Yaskawa INFORM job: DEMO_ROOF_UPPER_0625_3PAINT_40.JBI

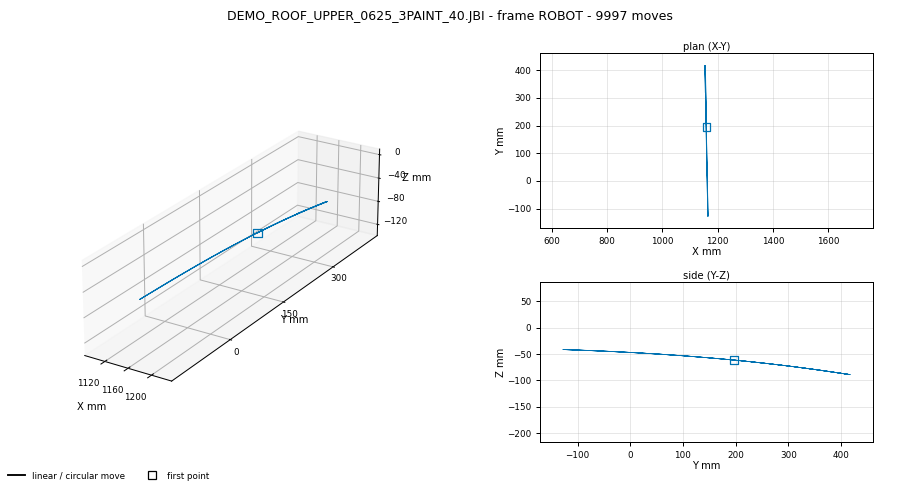
[picture p0: tool path of DEMO_ROOF_UPPER_0625_3PAINT_40.JBI in frame ROBOT, 9997 of 9997 moves have a stored position in this frame; points joined in program order, loops and branches not executed]
/JOB
//NAME DEMO_ROOF_UPPER_0625_3PAINT40
//POS
///NPOS 9997,0,0,0,0,0
///TOOL 0
///USER 0
///POSTYPE ROBOT
///RECTAN
///RCONF 1,0,0,0,0,0,0,0,0,0,0,0,0,0,0,0,0,0,0,0,0,0,0,0
C00000=1159.297,196.712,-61.157,-178.041,7.113,148.757
C00001=1159.293,196.961,-61.181,-178.039,7.115,148.757
C00002=1159.289,197.210,-61.205,-178.035,7.118,148.757
C00003=1159.284,197.459,-61.229,-178.033,7.120,148.756
C00004=1159.280,197.708,-61.253,-178.030,7.122,148.756
C00005=1159.275,197.956,-61.277,-178.027,7.124,148.756
C00006=1159.271,198.205,-61.300,-178.024,7.127,148.756
C00007=1159.265,198.454,-61.325,-178.022,7.129,148.756
C00008=1159.261,198.702,-61.349,-178.019,7.131,148.755
C00009=1159.257,198.952,-61.372,-178.016,7.134,148.755
C00010=1159.252,199.201,-61.396,-178.013,7.135,148.755
C00011=1159.248,199.450,-61.420,-178.011,7.138,148.755
C00012=1159.243,199.698,-61.445,-178.008,7.140,148.754
C00013=1159.238,199.947,-61.469,-178.005,7.143,148.754
C00014=1159.234,200.195,-61.493,-178.003,7.145,148.754
C00015=1159.229,200.444,-61.516,-177.999,7.147,148.754
C00016=1159.225,200.694,-61.541,-177.997,7.149,148.753
C00017=1159.220,200.942,-61.565,-177.994,7.152,148.753
C00018=1159.216,201.191,-61.588,-177.992,7.154,148.753
C00019=1159.211,201.439,-61.613,-177.989,7.156,148.753
C00020=1159.206,201.688,-61.637,-177.986,7.159,148.752
C00021=1159.202,201.937,-61.662,-177.983,7.161,148.752
C00022=1159.198,202.186,-61.685,-177.981,7.164,148.752
C00023=1159.192,202.435,-61.710,-177.978,7.165,148.752
C00024=1159.188,202.683,-61.734,-177.975,7.168,148.751
C00025=1159.184,202.933,-61.758,-177.973,7.170,148.751
C00026=1159.179,203.181,-61.783,-177.969,7.173,148.751
C00027=1159.175,203.430,-61.807,-177.967,7.175,148.751
C00028=1159.170,203.679,-61.830,-177.964,7.177,148.750
C00029=1159.165,203.928,-61.855,-177.962,7.179,148.750
C00030=1159.161,204.177,-61.879,-177.958,7.182,148.750
C00031=1159.157,204.425,-61.903,-177.956,7.184,148.750
C00032=1159.152,204.674,-61.928,-177.953,7.187,148.750
C00033=1159.148,204.923,-61.953,-177.951,7.189,148.749
C00034=1159.143,205.171,-61.977,-177.947,7.191,148.749
C00035=1159.138,205.420,-62.001,-177.945,7.193,148.749
C00036=1159.134,205.668,-62.025,-177.942,7.196,148.749
C00037=1159.129,205.918,-62.050,-177.940,7.198,148.749
C00038=1159.125,206.166,-62.075,-177.937,7.201,148.748
C00039=1159.120,206.415,-62.099,-177.934,7.203,148.748
C00040=1159.116,206.664,-62.124,-177.931,7.205,148.748
C00041=1159.111,206.913,-62.148,-177.929,7.208,148.748
C00042=1159.106,207.161,-62.172,-177.926,7.210,148.747
C00043=1159.101,207.410,-62.197,-177.923,7.212,148.747
C00044=1159.098,207.659,-62.221,-177.920,7.215,148.747
C00045=1159.093,207.907,-62.246,-177.918,7.217,148.747
C00046=1159.088,208.156,-62.270,-177.915,7.220,148.746
C00047=1159.083,208.406,-62.295,-177.913,7.222,148.746
C00048=1159.079,208.654,-62.319,-177.909,7.224,148.746
C00049=1159.074,208.903,-62.344,-177.907,7.226,148.746
C00050=1159.070,209.152,-62.368,-177.904,7.229,148.746
C00051=1159.065,209.400,-62.394,-177.902,7.231,148.745
C00052=1159.060,209.671,-62.420,-177.898,7.234,148.745
C00053=1159.055,209.942,-62.447,-177.895,7.236,148.745
C00054=1159.050,210.212,-62.474,-177.892,7.239,148.745
C00055=1159.046,210.483,-62.501,-177.889,7.242,148.744
C00056=1159.041,210.731,-62.525,-177.887,7.244,148.744
C00057=1159.037,210.980,-62.551,-177.884,7.246,148.744
C00058=1159.033,211.228,-62.575,-177.881,7.249,148.744
C00059=1159.027,211.477,-62.599,-177.878,7.251,148.744
C00060=1159.023,211.726,-62.624,-177.876,7.253,148.743
C00061=1159.019,211.974,-62.649,-177.873,7.256,148.743
C00062=1159.014,212.224,-62.674,-177.870,7.258,148.743
C00063=1159.009,212.472,-62.699,-177.867,7.261,148.743
C00064=1159.006,212.721,-62.724,-177.865,7.263,148.743
C00065=1159.001,212.970,-62.749,-177.862,7.266,148.742
C00066=1158.995,213.218,-62.773,-177.859,7.268,148.742
C00067=1158.992,213.467,-62.798,-177.857,7.270,148.742
C00068=1158.987,213.716,-62.823,-177.854,7.273,148.742
C00069=1158.982,213.965,-62.848,-177.851,7.275,148.742
C00070=1158.978,214.213,-62.873,-177.848,7.278,148.741
C00071=1158.974,214.462,-62.898,-177.846,7.280,148.741
C00072=1158.969,214.711,-62.923,-177.843,7.282,148.741
C00073=1158.965,214.959,-62.948,-177.840,7.284,148.741
C00074=1158.960,215.208,-62.972,-177.838,7.287,148.741
C00075=1158.956,215.457,-62.998,-177.834,7.290,148.740
C00076=1158.951,215.706,-63.023,-177.832,7.292,148.740
C00077=1158.947,215.954,-63.048,-177.829,7.295,148.740
C00078=1158.942,216.203,-63.073,-177.827,7.297,148.740
C00079=1158.938,216.452,-63.098,-177.823,7.299,148.739
C00080=1158.933,216.700,-63.123,-177.821,7.301,148.739
C00081=1158.928,216.949,-63.149,-177.819,7.304,148.739
C00082=1158.924,217.198,-63.173,-177.815,7.307,148.739
C00083=1158.920,217.446,-63.199,-177.813,7.309,148.739
C00084=1158.915,217.695,-63.223,-177.810,7.312,148.738
C00085=1158.910,217.944,-63.249,-177.808,7.314,148.738
C00086=1158.905,218.193,-63.274,-177.805,7.317,148.738
C00087=1158.902,218.441,-63.299,-177.802,7.319,148.738
C00088=1158.897,218.689,-63.324,-177.799,7.321,148.738
C00089=1158.892,218.939,-63.349,-177.796,7.324,148.738
C00090=1158.888,219.187,-63.375,-177.794,7.326,148.737
C00091=1158.883,219.436,-63.401,-177.791,7.329,148.737
C00092=1158.879,219.685,-63.426,-177.788,7.332,148.737
C00093=1158.874,219.933,-63.451,-177.786,7.334,148.737
C00094=1158.871,220.182,-63.476,-177.782,7.336,148.737
C00095=1158.865,220.430,-63.501,-177.780,7.338,148.736
C00096=1158.861,220.679,-63.527,-177.777,7.341,148.736
C00097=1158.857,220.928,-63.552,-177.774,7.344,148.736
C00098=1158.852,221.177,-63.577,-177.772,7.346,148.736
C00099=1158.848,221.425,-63.603,-177.769,7.349,148.736
C00100=1158.843,221.674,-63.628,-177.767,7.351,148.736
C00101=1158.839,221.922,-63.654,-177.764,7.354,148.735
C00102=1158.834,222.171,-63.680,-177.761,7.356,148.735
C00103=1158.829,222.420,-63.704,-177.758,7.358,148.735
C00104=1158.825,222.669,-63.730,-177.756,7.361,148.735
C00105=1158.821,222.918,-63.756,-177.752,7.364,148.735
C00106=1158.816,223.166,-63.781,-177.750,7.366,148.735
C00107=1158.812,223.414,-63.807,-177.747,7.369,148.734
C00108=1158.807,223.663,-63.832,-177.744,7.372,148.734
C00109=1158.802,223.912,-63.857,-177.742,7.374,148.734
C00110=1158.798,224.161,-63.883,-177.739,7.376,148.734
C00111=1158.793,224.409,-63.908,-177.736,7.378,148.734
C00112=1158.789,224.658,-63.934,-177.734,7.381,148.734
C00113=1158.785,224.906,-63.960,-177.730,7.384,148.733
C00114=1158.781,225.155,-63.986,-177.728,7.386,148.733
C00115=1158.776,225.403,-64.011,-177.725,7.389,148.733
C00116=1158.772,225.652,-64.037,-177.722,7.392,148.733
C00117=1158.767,225.901,-64.063,-177.720,7.394,148.733
C00118=1158.762,226.149,-64.088,-177.717,7.397,148.732
C00119=1158.758,226.398,-64.114,-177.714,7.399,148.732
C00120=1158.753,226.647,-64.140,-177.712,7.401,148.732
C00121=1158.748,226.895,-64.165,-177.709,7.404,148.732
C00122=1158.744,227.144,-64.191,-177.706,7.407,148.732
C00123=1158.740,227.393,-64.217,-177.704,7.409,148.732
C00124=1158.736,227.642,-64.243,-177.701,7.412,148.731
C00125=1158.731,227.890,-64.268,-177.698,7.415,148.731
C00126=1158.726,228.139,-64.294,-177.695,7.417,148.731
C00127=1158.722,228.388,-64.320,-177.693,7.420,148.731
C00128=1158.718,228.636,-64.346,-177.690,7.423,148.731
C00129=1158.713,228.884,-64.371,-177.687,7.424,148.731
C00130=1158.709,229.133,-64.398,-177.684,7.427,148.731
C00131=1158.705,229.381,-64.424,-177.682,7.430,148.730
C00132=1158.700,229.631,-64.450,-177.679,7.432,148.730
C00133=1158.695,229.879,-64.476,-177.676,7.435,148.730
C00134=1158.691,230.127,-64.501,-177.673,7.438,148.730
C00135=1158.686,230.376,-64.527,-177.671,7.440,148.730
C00136=1158.682,230.625,-64.554,-177.668,7.443,148.730
C00137=1158.677,230.874,-64.580,-177.665,7.446,148.729
C00138=1158.673,231.122,-64.605,-177.663,7.448,148.729
C00139=1158.668,231.370,-64.631,-177.660,7.450,148.729
C00140=1158.664,231.619,-64.658,-177.657,7.453,148.729
C00141=1158.660,231.868,-64.684,-177.654,7.456,148.729
C00142=1158.655,232.117,-64.709,-177.651,7.458,148.729
C00143=1158.651,232.365,-64.736,-177.649,7.461,148.728
C00144=1158.646,232.613,-64.762,-177.646,7.464,148.728
C00145=1158.642,232.862,-64.787,-177.644,7.466,148.728
C00146=1158.637,233.110,-64.815,-177.640,7.468,148.728
C00147=1158.633,233.359,-64.840,-177.638,7.471,148.728
C00148=1158.628,233.608,-64.866,-177.635,7.474,148.728
C00149=1158.624,233.857,-64.893,-177.633,7.476,148.728
C00150=1158.620,234.105,-64.919,-177.630,7.479,148.727
C00151=1158.615,234.354,-64.945,-177.627,7.482,148.727
C00152=1158.610,234.602,-64.971,-177.625,7.484,148.727
C00153=1158.606,234.851,-64.997,-177.622,7.487,148.727
C00154=1158.601,235.099,-65.024,-177.619,7.490,148.727
C00155=1158.597,235.348,-65.050,-177.616,7.493,148.727
C00156=1158.593,235.619,-65.079,-177.613,7.496,148.727
C00157=1158.587,235.892,-65.107,-177.610,7.498,148.726
C00158=1158.583,236.163,-65.136,-177.607,7.501,148.726
C00159=1158.578,236.434,-65.165,-177.604,7.504,148.726
C00160=1158.573,236.683,-65.191,-177.601,7.507,148.726
C00161=1158.569,236.932,-65.218,-177.599,7.509,148.726
C00162=1158.565,237.181,-65.244,-177.596,7.512,148.726
C00163=1158.560,237.429,-65.271,-177.593,7.515,148.726
C00164=1158.556,237.678,-65.297,-177.590,7.518,148.726
C00165=1158.551,237.926,-65.324,-177.588,7.519,148.725
C00166=1158.547,238.175,-65.350,-177.585,7.522,148.725
C00167=1158.542,238.424,-65.377,-177.582,7.525,148.725
C00168=1158.538,238.672,-65.403,-177.579,7.528,148.725
C00169=1158.534,238.920,-65.430,-177.577,7.530,148.725
C00170=1158.529,239.169,-65.456,-177.574,7.533,148.725
C00171=1158.525,239.418,-65.483,-177.571,7.536,148.725
C00172=1158.520,239.666,-65.510,-177.568,7.539,148.725
C00173=1158.516,239.915,-65.536,-177.566,7.541,148.724
C00174=1158.511,240.163,-65.563,-177.563,7.544,148.724
C00175=1158.507,240.412,-65.589,-177.560,7.546,148.724
C00176=1158.502,240.661,-65.616,-177.557,7.549,148.724
C00177=1158.498,240.909,-65.642,-177.555,7.552,148.724
C00178=1158.494,241.157,-65.669,-177.553,7.554,148.724
C00179=1158.489,241.406,-65.696,-177.550,7.557,148.724
C00180=1158.485,241.655,-65.722,-177.547,7.560,148.723
C00181=1158.480,241.903,-65.749,-177.544,7.562,148.723
C00182=1158.476,242.152,-65.776,-177.542,7.565,148.723
C00183=1158.472,242.400,-65.803,-177.539,7.568,148.723
C00184=1158.467,242.648,-65.830,-177.536,7.571,148.723
C00185=1158.462,242.897,-65.857,-177.533,7.574,148.723
C00186=1158.458,243.146,-65.882,-177.531,7.576,148.723
C00187=1158.453,243.394,-65.910,-177.528,7.579,148.723
C00188=1158.449,243.643,-65.937,-177.525,7.582,148.723
C00189=1158.445,243.891,-65.963,-177.522,7.585,148.722
C00190=1158.440,244.139,-65.990,-177.519,7.587,148.722
C00191=1158.436,244.389,-66.018,-177.517,7.590,148.722
C00192=1158.432,244.637,-66.044,-177.514,7.592,148.722
C00193=1158.428,244.885,-66.071,-177.511,7.595,148.722
C00194=1158.423,245.134,-66.098,-177.508,7.598,148.722
C00195=1158.418,245.382,-66.125,-177.506,7.600,148.722
C00196=1158.414,245.630,-66.152,-177.504,7.603,148.722
C00197=1158.410,245.879,-66.179,-177.501,7.606,148.722
C00198=1158.405,246.127,-66.206,-177.498,7.609,148.722
C00199=1158.401,246.377,-66.233,-177.495,7.612,148.721
C00200=1158.396,246.625,-66.260,-177.493,7.614,148.721
C00201=1158.392,246.873,-66.287,-177.490,7.617,148.721
C00202=1158.388,247.122,-66.314,-177.487,7.620,148.721
C00203=1158.383,247.370,-66.341,-177.484,7.623,148.721
C00204=1158.378,247.619,-66.368,-177.481,7.626,148.721
C00205=1158.374,247.867,-66.395,-177.479,7.628,148.721
C00206=1158.370,248.116,-66.423,-177.477,7.631,148.721
C00207=1158.366,248.364,-66.450,-177.474,7.634,148.721
C00208=1158.361,248.613,-66.477,-177.471,7.636,148.720
C00209=1158.357,248.861,-66.504,-177.468,7.639,148.720
C00210=1158.352,249.110,-66.531,-177.465,7.642,148.720
C00211=1158.347,249.358,-66.558,-177.463,7.644,148.720
C00212=1158.344,249.607,-66.586,-177.460,7.647,148.720
C00213=1158.339,249.855,-66.613,-177.457,7.650,148.720
C00214=1158.334,250.104,-66.640,-177.454,7.653,148.720
C00215=1158.330,250.352,-66.667,-177.452,7.656,148.720
C00216=1158.327,250.600,-66.695,-177.449,7.659,148.720
C00217=1158.322,250.849,-66.722,-177.447,7.661,148.720
C00218=1158.317,251.097,-66.749,-177.444,7.664,148.720
C00219=1158.313,251.346,-66.776,-177.441,7.667,148.719
C00220=1158.308,251.594,-66.804,-177.438,7.669,148.719
C00221=1158.304,251.843,-66.831,-177.435,7.672,148.719
C00222=1158.300,252.091,-66.858,-177.432,7.675,148.719
C00223=1158.295,252.339,-66.886,-177.430,7.677,148.719
C00224=1158.291,252.588,-66.913,-177.427,7.680,148.719
C00225=1158.287,252.837,-66.940,-177.425,7.683,148.719
C00226=1158.282,253.085,-66.968,-177.422,7.686,148.719
C00227=1158.278,253.333,-66.995,-177.419,7.689,148.719
C00228=1158.274,253.582,-67.023,-177.416,7.692,148.719
C00229=1158.269,253.830,-67.050,-177.414,7.695,148.719
C00230=1158.265,254.078,-67.078,-177.411,7.697,148.719
C00231=1158.261,254.327,-67.106,-177.409,7.700,148.719
C00232=1158.256,254.576,-67.134,-177.406,7.703,148.718
C00233=1158.251,254.824,-67.161,-177.403,7.706,148.718
C00234=1158.246,255.073,-67.188,-177.400,7.709,148.718
C00235=1158.243,255.321,-67.216,-177.398,7.712,148.718
C00236=1158.238,255.569,-67.244,-177.395,7.715,148.718
C00237=1158.234,255.818,-67.271,-177.393,7.717,148.718
C00238=1158.230,256.066,-67.299,-177.390,7.720,148.718
C00239=1158.225,256.315,-67.326,-177.387,7.723,148.718
C00240=1158.221,256.563,-67.354,-177.384,7.726,148.718
C00241=1158.216,256.812,-67.382,-177.381,7.729,148.718
C00242=1158.212,257.060,-67.410,-177.378,7.731,148.718
C00243=1158.208,257.309,-67.438,-177.376,7.734,148.718
C00244=1158.203,257.557,-67.465,-177.373,7.737,148.717
C00245=1158.199,257.805,-67.493,-177.371,7.739,148.717
C00246=1158.195,258.054,-67.520,-177.368,7.742,148.717
C00247=1158.190,258.302,-67.549,-177.365,7.745,148.717
C00248=1158.185,258.550,-67.576,-177.362,7.748,148.717
C00249=1158.182,258.799,-67.605,-177.360,7.751,148.717
C00250=1158.177,259.047,-67.632,-177.357,7.754,148.717
C00251=1158.173,259.296,-67.660,-177.354,7.757,148.717
C00252=1158.168,259.544,-67.688,-177.351,7.760,148.717
C00253=1158.164,259.792,-67.715,-177.349,7.763,148.717
C00254=1158.160,260.041,-67.743,-177.347,7.766,148.717
C00255=1158.155,260.289,-67.771,-177.344,7.768,148.717
C00256=1158.151,260.538,-67.800,-177.341,7.771,148.717
C00257=1158.147,260.786,-67.828,-177.338,7.774,148.717
C00258=1158.143,261.035,-67.855,-177.336,7.777,148.717
C00259=1158.138,261.283,-67.883,-177.333,7.780,148.717
C00260=1158.133,261.556,-67.914,-177.330,7.783,148.717
C00261=1158.128,261.830,-67.945,-177.327,7.786,148.717
C00262=1158.124,262.102,-67.976,-177.324,7.790,148.717
C00263=1158.119,262.376,-68.007,-177.321,7.793,148.716
C00264=1158.114,262.624,-68.035,-177.318,7.796,148.716
C00265=1158.110,262.873,-68.063,-177.316,7.799,148.716
C00266=1158.106,263.121,-68.090,-177.313,7.802,148.716
C00267=1158.101,263.370,-68.119,-177.310,7.805,148.716
C00268=1158.097,263.618,-68.147,-177.307,7.808,148.716
C00269=1158.093,263.866,-68.175,-177.305,7.811,148.716
C00270=1158.088,264.115,-68.204,-177.302,7.813,148.716
C00271=1158.084,264.363,-68.232,-177.300,7.816,148.716
C00272=1158.079,264.611,-68.260,-177.297,7.819,148.716
C00273=1158.075,264.860,-68.288,-177.294,7.822,148.716
C00274=1158.070,265.108,-68.317,-177.291,7.824,148.716
C00275=1158.067,265.357,-68.345,-177.289,7.827,148.716
C00276=1158.061,265.605,-68.373,-177.286,7.830,148.716
C00277=1158.058,265.853,-68.402,-177.283,7.833,148.716
C00278=1158.054,266.101,-68.430,-177.280,7.836,148.716
C00279=1158.049,266.350,-68.458,-177.278,7.840,148.716
C00280=1158.045,266.598,-68.487,-177.275,7.842,148.716
C00281=1158.040,266.846,-68.515,-177.272,7.845,148.716
C00282=1158.037,267.095,-68.543,-177.270,7.848,148.716
C00283=1158.032,267.343,-68.571,-177.267,7.851,148.716
C00284=1158.027,267.592,-68.600,-177.265,7.853,148.715
C00285=1158.024,267.840,-68.629,-177.262,7.856,148.715
C00286=1158.018,268.088,-68.657,-177.259,7.859,148.715
C00287=1158.015,268.337,-68.686,-177.256,7.862,148.715
C00288=1158.010,268.585,-68.714,-177.254,7.866,148.715
C00289=1158.006,268.833,-68.742,-177.251,7.869,148.715
C00290=1158.002,269.082,-68.772,-177.249,7.871,148.715
C00291=1157.997,269.330,-68.799,-177.246,7.874,148.715
C00292=1157.993,269.579,-68.828,-177.243,7.877,148.715
C00293=1157.988,269.826,-68.857,-177.240,7.880,148.715
C00294=1157.984,270.075,-68.885,-177.238,7.883,148.715
C00295=1157.980,270.324,-68.914,-177.235,7.886,148.715
C00296=1157.976,270.571,-68.942,-177.232,7.890,148.715
C00297=1157.971,270.820,-68.971,-177.230,7.892,148.715
C00298=1157.967,271.069,-69.000,-177.227,7.895,148.715
C00299=1157.963,271.316,-69.028,-177.224,7.898,148.715
C00300=1157.958,271.565,-69.057,-177.221,7.901,148.715
C00301=1157.954,271.814,-69.086,-177.219,7.904,148.715
C00302=1157.950,272.061,-69.114,-177.216,7.907,148.715
C00303=1157.945,272.310,-69.143,-177.214,7.910,148.715
C00304=1157.941,272.558,-69.173,-177.211,7.913,148.715
C00305=1157.937,272.806,-69.200,-177.208,7.916,148.715
C00306=1157.932,273.055,-69.229,-177.205,7.919,148.715
C00307=1157.928,273.303,-69.259,-177.203,7.921,148.715
C00308=1157.924,273.552,-69.287,-177.200,7.924,148.715
C00309=1157.920,273.799,-69.316,-177.198,7.928,148.715
C00310=1157.915,274.048,-69.345,-177.195,7.931,148.715
C00311=1157.911,274.296,-69.374,-177.192,7.934,148.715
C00312=1157.906,274.544,-69.403,-177.190,7.937,148.715
C00313=1157.902,274.792,-69.431,-177.187,7.940,148.715
C00314=1157.898,275.041,-69.461,-177.185,7.943,148.715
C00315=1157.894,275.290,-69.489,-177.182,7.946,148.715
C00316=1157.889,275.537,-69.519,-177.179,7.949,148.715
C00317=1157.884,275.786,-69.547,-177.176,7.952,148.715
C00318=1157.881,276.034,-69.576,-177.174,7.955,148.715
C00319=1157.877,276.282,-69.606,-177.171,7.958,148.715
C00320=1157.872,276.531,-69.634,-177.169,7.961,148.715
C00321=1157.868,276.779,-69.663,-177.166,7.964,148.715
C00322=1157.863,277.027,-69.693,-177.163,7.967,148.715
C00323=1157.859,277.276,-69.722,-177.160,7.970,148.715
C00324=1157.855,277.524,-69.750,-177.158,7.973,148.715
C00325=1157.851,277.771,-69.780,-177.155,7.976,148.715
C00326=1157.846,278.020,-69.809,-177.152,7.979,148.715
C00327=1157.842,278.269,-69.838,-177.150,7.982,148.715
C00328=1157.838,278.517,-69.867,-177.147,7.985,148.715
C00329=1157.834,278.765,-69.897,-177.145,7.988,148.715
C00330=1157.829,279.013,-69.926,-177.142,7.991,148.715
C00331=1157.824,279.262,-69.954,-177.139,7.994,148.715
C00332=1157.820,279.510,-69.984,-177.137,7.997,148.715
C00333=1157.817,279.758,-70.013,-177.134,8.000,148.715
C00334=1157.813,280.006,-70.042,-177.131,8.003,148.715
C00335=1157.808,280.254,-70.072,-177.128,8.006,148.715
C00336=1157.804,280.503,-70.101,-177.126,8.009,148.715
C00337=1157.800,280.751,-70.131,-177.123,8.012,148.715
C00338=1157.795,280.999,-70.159,-177.121,8.015,148.715
C00339=1157.791,281.247,-70.188,-177.118,8.018,148.715
C00340=1157.787,281.496,-70.218,-177.116,8.022,148.715
C00341=1157.782,281.744,-70.247,-177.113,8.024,148.715
C00342=1157.778,281.992,-70.277,-177.110,8.027,148.715
C00343=1157.774,282.240,-70.306,-177.107,8.031,148.715
C00344=1157.769,282.489,-70.336,-177.104,8.034,148.715
C00345=1157.765,282.737,-70.366,-177.102,8.037,148.715
C00346=1157.761,282.986,-70.395,-177.099,8.040,148.715
C00347=1157.756,283.233,-70.424,-177.097,8.044,148.715
C00348=1157.752,283.481,-70.454,-177.094,8.047,148.715
C00349=1157.748,283.730,-70.483,-177.091,8.050,148.715
C00350=1157.743,283.978,-70.513,-177.088,8.053,148.715
C00351=1157.739,284.226,-70.542,-177.086,8.056,148.715
C00352=1157.735,284.474,-70.572,-177.083,8.059,148.715
C00353=1157.731,284.723,-70.601,-177.080,8.062,148.715
C00354=1157.727,284.971,-70.630,-177.078,8.065,148.715
C00355=1157.722,285.219,-70.661,-177.075,8.068,148.715
C00356=1157.718,285.467,-70.691,-177.073,8.071,148.715
C00357=1157.714,285.715,-70.720,-177.070,8.074,148.715
C00358=1157.709,285.964,-70.750,-177.068,8.077,148.715
C00359=1157.705,286.212,-70.779,-177.065,8.080,148.715
C00360=1157.701,286.460,-70.808,-177.062,8.083,148.715
C00361=1157.697,286.708,-70.839,-177.060,8.086,148.715
C00362=1157.692,286.956,-70.869,-177.057,8.089,148.715
C00363=1157.688,287.205,-70.898,-177.055,8.093,148.716
C00364=1157.684,287.480,-70.931,-177.051,8.096,148.716
C00365=1157.679,287.755,-70.964,-177.049,8.099,148.716
C00366=1157.674,288.030,-70.997,-177.045,8.103,148.716
C00367=1157.669,288.305,-71.030,-177.043,8.106,148.716
C00368=1157.665,288.553,-71.060,-177.040,8.109,148.716
C00369=1157.660,288.801,-71.090,-177.037,8.112,148.716
C00370=1157.656,289.050,-71.120,-177.034,8.116,148.716
C00371=1157.652,289.297,-71.150,-177.032,8.119,148.716
C00372=1157.648,289.545,-71.179,-177.029,8.123,148.716
C00373=1157.644,289.795,-71.210,-177.027,8.126,148.716
C00374=1157.640,290.042,-71.240,-177.024,8.128,148.716
C00375=1157.636,290.291,-71.269,-177.022,8.132,148.716
C00376=1157.631,290.539,-71.300,-177.019,8.135,148.716
C00377=1157.627,290.787,-71.330,-177.016,8.138,148.716
C00378=1157.623,291.035,-71.359,-177.014,8.141,148.716
C00379=1157.618,291.283,-71.390,-177.011,8.144,148.716
C00380=1157.614,291.531,-71.419,-177.009,8.147,148.716
C00381=1157.610,291.779,-71.449,-177.006,8.150,148.716
C00382=1157.605,292.028,-71.479,-177.003,8.153,148.716
C00383=1157.601,292.275,-71.510,-177.000,8.157,148.716
C00384=1157.598,292.524,-71.539,-176.998,8.160,148.716
C00385=1157.593,292.772,-71.570,-176.995,8.163,148.717
C00386=1157.589,293.020,-71.600,-176.992,8.166,148.717
C00387=1157.584,293.268,-71.630,-176.990,8.169,148.717
C00388=1157.580,293.516,-71.661,-176.987,8.173,148.717
C00389=1157.575,293.765,-71.691,-176.985,8.176,148.717
C00390=1157.571,294.012,-71.721,-176.982,8.179,148.717
C00391=1157.568,294.261,-71.751,-176.980,8.182,148.717
C00392=1157.563,294.509,-71.781,-176.977,8.185,148.717
C00393=1157.559,294.757,-71.812,-176.975,8.188,148.717
C00394=1157.554,295.005,-71.842,-176.971,8.192,148.717
C00395=1157.551,295.253,-71.872,-176.969,8.195,148.717
C00396=1157.546,295.501,-71.903,-176.966,8.198,148.717
C00397=1157.542,295.750,-71.932,-176.964,8.201,148.717
C00398=1157.538,295.998,-71.963,-176.961,8.204,148.717
C00399=1157.534,296.246,-71.993,-176.959,8.208,148.717
C00400=1157.529,296.494,-72.024,-176.956,8.211,148.717
C00401=1157.525,296.742,-72.053,-176.953,8.213,148.717
C00402=1157.521,296.990,-72.085,-176.951,8.217,148.718
C00403=1157.517,297.238,-72.115,-176.948,8.220,148.718
C00404=1157.513,297.486,-72.146,-176.945,8.224,148.718
C00405=1157.508,297.734,-72.176,-176.943,8.227,148.718
C00406=1157.504,297.983,-72.206,-176.940,8.230,148.718
C00407=1157.500,298.231,-72.237,-176.937,8.233,148.718
C00408=1157.496,298.479,-72.267,-176.935,8.236,148.718
C00409=1157.491,298.727,-72.298,-176.932,8.239,148.718
C00410=1157.487,298.975,-72.329,-176.930,8.243,148.718
C00411=1157.483,299.223,-72.359,-176.927,8.246,148.718
C00412=1157.479,299.471,-72.390,-176.924,8.250,148.718
C00413=1157.474,299.719,-72.421,-176.922,8.253,148.718
C00414=1157.471,299.968,-72.450,-176.919,8.256,148.719
C00415=1157.466,300.216,-72.481,-176.917,8.259,148.718
C00416=1157.461,300.464,-72.512,-176.914,8.262,148.719
C00417=1157.458,300.711,-72.542,-176.912,8.265,148.719
C00418=1157.454,300.960,-72.573,-176.909,8.268,148.719
C00419=1157.449,301.208,-72.604,-176.906,8.271,148.719
C00420=1157.445,301.456,-72.634,-176.904,8.275,148.719
C00421=1157.441,301.704,-72.665,-176.901,8.278,148.719
C00422=1157.436,301.952,-72.696,-176.899,8.282,148.719
C00423=1157.432,302.200,-72.728,-176.896,8.285,148.719
C00424=1157.429,302.448,-72.758,-176.893,8.288,148.719
C00425=1157.424,302.696,-72.789,-176.891,8.291,148.719
C00426=1157.420,302.944,-72.820,-176.888,8.294,148.719
C00427=1157.416,303.192,-72.851,-176.885,8.298,148.719
C00428=1157.412,303.440,-72.881,-176.883,8.301,148.720
C00429=1157.407,303.688,-72.912,-176.880,8.304,148.720
C00430=1157.403,303.937,-72.943,-176.878,8.307,148.720
C00431=1157.398,304.185,-72.974,-176.875,8.311,148.720
C00432=1157.394,304.432,-73.005,-176.873,8.314,148.720
C00433=1157.390,304.681,-73.036,-176.870,8.318,148.720
C00434=1157.386,304.928,-73.066,-176.867,8.321,148.720
C00435=1157.382,305.177,-73.098,-176.865,8.324,148.720
C00436=1157.378,305.424,-73.129,-176.862,8.327,148.720
C00437=1157.373,305.672,-73.160,-176.860,8.330,148.720
C00438=1157.369,305.921,-73.191,-176.857,8.333,148.721
C00439=1157.365,306.169,-73.222,-176.854,8.337,148.721
C00440=1157.361,306.417,-73.254,-176.852,8.341,148.721
C00441=1157.356,306.665,-73.284,-176.849,8.344,148.721
C00442=1157.353,306.913,-73.314,-176.847,8.347,148.721
C00443=1157.349,307.161,-73.346,-176.844,8.350,148.721
C00444=1157.344,307.409,-73.377,-176.842,8.353,148.721
C00445=1157.340,307.657,-73.408,-176.839,8.357,148.721
C00446=1157.336,307.905,-73.440,-176.836,8.360,148.721
C00447=1157.332,308.153,-73.471,-176.834,8.363,148.722
C00448=1157.327,308.401,-73.502,-176.831,8.366,148.722
C00449=1157.323,308.648,-73.533,-176.829,8.370,148.722
C00450=1157.319,308.897,-73.564,-176.826,8.373,148.722
C00451=1157.315,309.144,-73.596,-176.823,8.377,148.722
C00452=1157.311,309.393,-73.627,-176.821,8.380,148.722
C00453=1157.306,309.640,-73.658,-176.818,8.383,148.722
C00454=1157.302,309.889,-73.689,-176.816,8.386,148.722
C00455=1157.298,310.136,-73.721,-176.813,8.389,148.722
C00456=1157.294,310.385,-73.752,-176.810,8.393,148.723
C00457=1157.290,310.632,-73.783,-176.808,8.397,148.723
C00458=1157.286,310.881,-73.815,-176.805,8.400,148.723
C00459=1157.281,311.128,-73.846,-176.803,8.403,148.723
C00460=1157.277,311.377,-73.877,-176.800,8.406,148.723
C00461=1157.273,311.624,-73.909,-176.797,8.410,148.723
C00462=1157.269,311.873,-73.941,-176.795,8.413,148.723
C00463=1157.265,312.120,-73.971,-176.792,8.416,148.723
C00464=1157.260,312.369,-74.004,-176.789,8.419,148.723
C00465=1157.256,312.617,-74.035,-176.787,8.423,148.724
C00466=1157.252,312.865,-74.066,-176.784,8.427,148.724
C00467=1157.248,313.113,-74.098,-176.782,8.430,148.724
C00468=1157.243,313.390,-74.133,-176.779,8.433,148.724
C00469=1157.239,313.668,-74.168,-176.776,8.437,148.724
C00470=1157.234,313.945,-74.204,-176.773,8.441,148.724
C00471=1157.229,314.222,-74.239,-176.770,8.445,148.724
C00472=1157.225,314.470,-74.271,-176.768,8.448,148.725
C00473=1157.221,314.718,-74.303,-176.765,8.451,148.725
C00474=1157.217,314.966,-74.334,-176.763,8.454,148.725
C00475=1157.212,315.214,-74.366,-176.760,8.458,148.725
C00476=1157.209,315.462,-74.398,-176.757,8.462,148.725
C00477=1157.204,315.709,-74.429,-176.755,8.465,148.725
C00478=1157.201,315.957,-74.461,-176.753,8.468,148.725
C00479=1157.196,316.206,-74.493,-176.750,8.471,148.726
C00480=1157.192,316.454,-74.524,-176.747,8.475,148.726
C00481=1157.188,316.702,-74.556,-176.745,8.478,148.726
C00482=1157.184,316.950,-74.588,-176.742,8.482,148.726
C00483=1157.180,317.197,-74.619,-176.739,8.485,148.726
C00484=1157.175,317.445,-74.652,-176.737,8.488,148.726
C00485=1157.172,317.693,-74.684,-176.734,8.492,148.726
C00486=1157.167,317.941,-74.715,-176.732,8.495,148.727
C00487=1157.163,318.189,-74.747,-176.729,8.498,148.727
C00488=1157.159,318.437,-74.779,-176.727,8.502,148.727
C00489=1157.155,318.684,-74.811,-176.724,8.506,148.727
C00490=1157.151,318.933,-74.843,-176.722,8.509,148.727
C00491=1157.147,319.181,-74.875,-176.719,8.512,148.727
C00492=1157.143,319.428,-74.907,-176.717,8.515,148.727
C00493=1157.138,319.677,-74.939,-176.714,8.519,148.728
C00494=1157.134,319.925,-74.971,-176.711,8.523,148.728
C00495=1157.131,320.173,-75.003,-176.709,8.526,148.728
C00496=1157.126,320.420,-75.035,-176.706,8.529,148.728
C00497=1157.122,320.668,-75.067,-176.704,8.533,148.728
C00498=1157.118,320.916,-75.098,-176.701,8.536,148.728
C00499=1157.114,321.165,-75.131,-176.698,8.539,148.728
C00500=1157.109,321.412,-75.162,-176.696,8.542,148.729
C00501=1157.105,321.660,-75.196,-176.693,8.547,148.729
C00502=1157.102,321.908,-75.227,-176.691,8.550,148.729
C00503=1157.098,322.156,-75.259,-176.688,8.553,148.729
C00504=1157.093,322.403,-75.291,-176.686,8.556,148.729
C00505=1157.089,322.652,-75.323,-176.683,8.560,148.729
C00506=1157.085,322.899,-75.356,-176.681,8.563,148.730
C00507=1157.081,323.147,-75.388,-176.678,8.567,148.730
C00508=1157.076,323.395,-75.420,-176.676,8.570,148.730
C00509=1157.073,323.643,-75.452,-176.673,8.574,148.730
C00510=1157.068,323.891,-75.485,-176.670,8.577,148.730
C00511=1157.065,324.139,-75.517,-176.668,8.580,148.730
C00512=1157.060,324.387,-75.549,-176.665,8.584,148.731
C00513=1157.056,324.634,-75.582,-176.663,8.588,148.731
C00514=1157.052,324.882,-75.614,-176.660,8.591,148.731
C00515=1157.048,325.130,-75.646,-176.658,8.594,148.731
C00516=1157.044,325.378,-75.679,-176.655,8.598,148.731
C00517=1157.040,325.626,-75.711,-176.653,8.601,148.732
C00518=1157.036,325.874,-75.743,-176.650,8.605,148.732
C00519=1157.031,326.121,-75.776,-176.647,8.609,148.732
C00520=1157.027,326.369,-75.808,-176.645,8.612,148.732
C00521=1157.023,326.617,-75.841,-176.642,8.615,148.732
C00522=1157.020,326.865,-75.873,-176.640,8.618,148.732
C00523=1157.015,327.114,-75.905,-176.637,8.622,148.733
C00524=1157.011,327.361,-75.939,-176.635,8.626,148.733
C00525=1157.007,327.609,-75.970,-176.633,8.629,148.733
C00526=1157.003,327.856,-76.003,-176.630,8.633,148.733
C00527=1156.998,328.105,-76.036,-176.627,8.636,148.733
C00528=1156.995,328.352,-76.068,-176.625,8.639,148.733
C00529=1156.991,328.600,-76.101,-176.622,8.643,148.734
C00530=1156.986,328.848,-76.134,-176.619,8.647,148.734
C00531=1156.983,329.096,-76.166,-176.617,8.650,148.734
C00532=1156.978,329.344,-76.199,-176.615,8.653,148.734
C00533=1156.974,329.592,-76.232,-176.612,8.657,148.734
C00534=1156.970,329.840,-76.264,-176.610,8.661,148.735
C00535=1156.966,330.087,-76.297,-176.607,8.664,148.735
C00536=1156.962,330.335,-76.330,-176.604,8.668,148.735
C00537=1156.957,330.583,-76.362,-176.602,8.671,148.735
C00538=1156.954,330.830,-76.395,-176.599,8.674,148.735
C00539=1156.950,331.078,-76.428,-176.597,8.678,148.736
C00540=1156.945,331.326,-76.460,-176.594,8.682,148.736
C00541=1156.941,331.574,-76.494,-176.592,8.685,148.736
C00542=1156.938,331.821,-76.526,-176.589,8.689,148.736
C00543=1156.933,332.069,-76.559,-176.587,8.692,148.736
C00544=1156.929,332.318,-76.592,-176.584,8.696,148.737
C00545=1156.925,332.565,-76.625,-176.581,8.700,148.737
C00546=1156.921,332.813,-76.658,-176.579,8.703,148.737
C00547=1156.917,333.061,-76.691,-176.577,8.706,148.737
C00548=1156.913,333.308,-76.724,-176.574,8.710,148.737
C00549=1156.909,333.556,-76.756,-176.571,8.713,148.737
C00550=1156.905,333.804,-76.789,-176.569,8.717,148.738
C00551=1156.900,334.052,-76.823,-176.566,8.721,148.738
C00552=1156.896,334.300,-76.856,-176.564,8.724,148.738
C00553=1156.892,334.547,-76.889,-176.561,8.727,148.738
C00554=1156.888,334.795,-76.922,-176.559,8.731,148.739
C00555=1156.885,335.043,-76.955,-176.556,8.735,148.739
C00556=1156.880,335.290,-76.988,-176.554,8.738,148.739
C00557=1156.876,335.538,-77.021,-176.551,8.742,148.739
C00558=1156.872,335.786,-77.054,-176.549,8.745,148.739
C00559=1156.868,336.034,-77.086,-176.546,8.749,148.740
C00560=1156.864,336.282,-77.120,-176.544,8.753,148.740
C00561=1156.860,336.530,-77.153,-176.541,8.756,148.740
C00562=1156.856,336.778,-77.186,-176.539,8.759,148.740
C00563=1156.852,337.025,-77.220,-176.536,8.763,148.741
C00564=1156.848,337.273,-77.253,-176.534,8.767,148.741
C00565=1156.844,337.521,-77.286,-176.531,8.770,148.741
C00566=1156.840,337.768,-77.320,-176.528,8.774,148.741
C00567=1156.836,338.016,-77.353,-176.526,8.777,148.741
C00568=1156.831,338.264,-77.386,-176.523,8.781,148.742
C00569=1156.827,338.511,-77.419,-176.521,8.785,148.742
C00570=1156.823,338.759,-77.452,-176.519,8.788,148.742
C00571=1156.820,339.008,-77.486,-176.516,8.792,148.742
C00572=1156.815,339.287,-77.523,-176.513,8.796,148.743
C00573=1156.810,339.567,-77.561,-176.510,8.800,148.743
C00574=1156.805,339.847,-77.599,-176.508,8.804,148.743
C00575=1156.801,340.127,-77.637,-176.505,8.808,148.743
C00576=1156.797,340.375,-77.670,-176.502,8.812,148.744
C00577=1156.793,340.622,-77.703,-176.500,8.815,148.744
C00578=1156.789,340.870,-77.737,-176.497,8.819,148.744
C00579=1156.785,341.117,-77.770,-176.495,8.823,148.744
C00580=1156.780,341.365,-77.804,-176.493,8.826,148.745
C00581=1156.776,341.614,-77.837,-176.490,8.830,148.745
C00582=1156.773,341.861,-77.871,-176.487,8.833,148.745
C00583=1156.768,342.109,-77.904,-176.484,8.837,148.745
C00584=1156.764,342.356,-77.938,-176.482,8.841,148.745
C00585=1156.760,342.603,-77.972,-176.480,8.844,148.746
C00586=1156.756,342.851,-78.005,-176.477,8.848,148.746
C00587=1156.752,343.099,-78.040,-176.475,8.851,148.746
C00588=1156.748,343.347,-78.073,-176.472,8.856,148.746
C00589=1156.744,343.595,-78.106,-176.469,8.859,148.747
C00590=1156.740,343.842,-78.140,-176.467,8.862,148.747
C00591=1156.736,344.091,-78.174,-176.465,8.866,148.747
C00592=1156.732,344.338,-78.208,-176.462,8.870,148.747
C00593=1156.728,344.585,-78.241,-176.459,8.874,148.748
C00594=1156.724,344.833,-78.275,-176.457,8.877,148.748
C00595=1156.719,345.081,-78.308,-176.455,8.880,148.748
C00596=1156.716,345.328,-78.343,-176.452,8.885,148.748
C00597=1156.712,345.576,-78.376,-176.450,8.888,148.749
C00598=1156.707,345.824,-78.410,-176.447,8.892,148.749
C00599=1156.703,346.071,-78.443,-176.445,8.896,148.749
C00600=1156.700,346.319,-78.478,-176.442,8.900,148.750
C00601=1156.696,346.567,-78.511,-176.440,8.903,148.750
C00602=1156.691,346.814,-78.545,-176.437,8.906,148.750
C00603=1156.688,347.063,-78.579,-176.434,8.910,148.750
C00604=1156.684,347.310,-78.613,-176.432,8.914,148.750
C00605=1156.679,347.557,-78.647,-176.429,8.918,148.751
C00606=1156.676,347.806,-78.681,-176.427,8.921,148.751
C00607=1156.671,348.053,-78.715,-176.424,8.925,148.751
C00608=1156.667,348.300,-78.749,-176.422,8.929,148.752
C00609=1156.663,348.548,-78.782,-176.420,8.932,148.752
C00610=1156.659,348.796,-78.817,-176.417,8.936,148.752
C00611=1156.655,349.043,-78.851,-176.415,8.939,148.752
C00612=1156.651,349.290,-78.885,-176.412,8.944,148.753
C00613=1156.647,349.539,-78.919,-176.410,8.947,148.753
C00614=1156.644,349.786,-78.953,-176.407,8.951,148.753
C00615=1156.640,350.034,-78.988,-176.405,8.954,148.753
C00616=1156.636,350.281,-79.021,-176.402,8.958,148.754
C00617=1156.631,350.529,-79.055,-176.400,8.962,148.754
C00618=1156.628,350.777,-79.089,-176.397,8.966,148.754
C00619=1156.623,351.025,-79.124,-176.395,8.969,148.755
C00620=1156.619,351.272,-79.158,-176.392,8.973,148.755
C00621=1156.615,351.520,-79.193,-176.390,8.977,148.755
C00622=1156.611,351.767,-79.227,-176.388,8.980,148.755
C00623=1156.607,352.015,-79.261,-176.385,8.985,148.756
C00624=1156.603,352.263,-79.294,-176.382,8.988,148.756
C00625=1156.599,352.510,-79.329,-176.380,8.992,148.756
C00626=1156.596,352.758,-79.363,-176.378,8.995,148.757
C00627=1156.591,353.005,-79.398,-176.375,9.000,148.757
C00628=1156.588,353.253,-79.432,-176.372,9.003,148.757
C00629=1156.583,353.501,-79.466,-176.370,9.007,148.757
C00630=1156.579,353.749,-79.501,-176.368,9.011,148.758
C00631=1156.575,353.996,-79.535,-176.365,9.015,148.758
C00632=1156.571,354.243,-79.570,-176.363,9.018,148.758
C00633=1156.568,354.491,-79.604,-176.360,9.022,148.758
C00634=1156.563,354.738,-79.638,-176.358,9.026,148.759
C00635=1156.559,354.987,-79.673,-176.355,9.030,148.759
C00636=1156.555,355.233,-79.708,-176.353,9.033,148.759
C00637=1156.552,355.481,-79.742,-176.350,9.037,148.760
C00638=1156.548,355.728,-79.776,-176.348,9.041,148.760
C00639=1156.544,355.976,-79.811,-176.345,9.045,148.760
C00640=1156.539,356.224,-79.846,-176.343,9.048,148.760
C00641=1156.536,356.472,-79.880,-176.340,9.052,148.761
C00642=1156.531,356.719,-79.914,-176.338,9.056,148.761
C00643=1156.528,356.967,-79.950,-176.335,9.060,148.761
C00644=1156.524,357.214,-79.984,-176.333,9.063,148.762
C00645=1156.520,357.462,-80.019,-176.330,9.068,148.762
C00646=1156.515,357.709,-80.053,-176.328,9.071,148.762
C00647=1156.511,357.957,-80.088,-176.325,9.075,148.763
C00648=1156.508,358.204,-80.123,-176.323,9.079,148.763
C00649=1156.504,358.452,-80.157,-176.320,9.083,148.763
C00650=1156.500,358.700,-80.192,-176.318,9.086,148.764
C00651=1156.496,358.947,-80.227,-176.315,9.090,148.764
C00652=1156.492,359.195,-80.262,-176.312,9.094,148.764
C00653=1156.488,359.442,-80.296,-176.311,9.098,148.765
C00654=1156.484,359.690,-80.332,-176.308,9.102,148.765
C00655=1156.480,359.937,-80.366,-176.305,9.105,148.765
C00656=1156.476,360.185,-80.400,-176.303,9.110,148.766
C00657=1156.473,360.432,-80.436,-176.301,9.113,148.766
C00658=1156.468,360.680,-80.470,-176.298,9.117,148.766
C00659=1156.464,360.927,-80.506,-176.295,9.122,148.767
C00660=1156.460,361.175,-80.540,-176.293,9.125,148.767
C00661=1156.457,361.423,-80.575,-176.290,9.129,148.767
C00662=1156.453,361.670,-80.610,-176.288,9.133,148.767
C00663=1156.448,361.917,-80.645,-176.285,9.137,148.768
C00664=1156.445,362.165,-80.680,-176.283,9.141,148.768
C00665=1156.441,362.413,-80.715,-176.281,9.144,148.768
C00666=1156.437,362.660,-80.750,-176.278,9.148,148.769
C00667=1156.433,362.908,-80.785,-176.276,9.152,148.769
C00668=1156.428,363.155,-80.820,-176.273,9.156,148.769
C00669=1156.425,363.402,-80.855,-176.270,9.161,148.770
C00670=1156.421,363.650,-80.890,-176.268,9.164,148.770
C00671=1156.417,363.897,-80.925,-176.265,9.168,148.770
C00672=1156.413,364.145,-80.960,-176.263,9.172,148.771
C00673=1156.410,364.392,-80.996,-176.260,9.176,148.771
C00674=1156.406,364.640,-81.031,-176.258,9.180,148.771
C00675=1156.401,364.887,-81.066,-176.256,9.183,148.772
C00676=1156.397,365.171,-81.106,-176.253,9.189,148.772
C00677=1156.393,365.453,-81.146,-176.250,9.193,148.773
C00678=1156.388,365.736,-81.187,-176.247,9.197,148.773
C00679=1156.384,366.019,-81.227,-176.245,9.201,148.773
C00680=1156.380,366.266,-81.262,-176.242,9.206,148.774
C00681=1156.376,366.513,-81.297,-176.239,9.210,148.774
C00682=1156.372,366.761,-81.332,-176.238,9.214,148.775
C00683=1156.368,367.009,-81.368,-176.235,9.218,148.775
C00684=1156.363,367.256,-81.404,-176.233,9.221,148.775
C00685=1156.360,367.503,-81.439,-176.230,9.226,148.776
C00686=1156.356,367.751,-81.475,-176.227,9.230,148.776
C00687=1156.352,367.999,-81.510,-176.226,9.233,148.776
C00688=1156.348,368.246,-81.545,-176.223,9.238,148.777
C00689=1156.344,368.493,-81.580,-176.221,9.241,148.777
C00690=1156.340,368.741,-81.616,-176.218,9.245,148.778
C00691=1156.337,368.988,-81.651,-176.216,9.250,148.778
C00692=1156.333,369.236,-81.687,-176.214,9.253,148.779
C00693=1156.328,369.483,-81.723,-176.211,9.258,148.779
C00694=1156.324,369.730,-81.758,-176.210,9.261,148.779
C00695=1156.321,369.978,-81.794,-176.207,9.266,148.780
C00696=1156.317,370.225,-81.829,-176.205,9.269,148.780
C00697=1156.313,370.473,-81.865,-176.202,9.274,148.781
C00698=1156.309,370.720,-81.900,-176.200,9.277,148.781
C00699=1156.305,370.968,-81.936,-176.198,9.282,148.781
C00700=1156.301,371.215,-81.972,-176.196,9.285,148.782
C00701=1156.297,371.463,-82.007,-176.194,9.290,148.782
C00702=1156.294,371.710,-82.043,-176.192,9.293,148.783
C00703=1156.290,371.958,-82.078,-176.190,9.298,148.783
C00704=1156.285,372.205,-82.114,-176.188,9.301,148.784
C00705=1156.281,372.452,-82.150,-176.185,9.306,148.784
C00706=1156.278,372.700,-82.185,-176.183,9.309,148.785
C00707=1156.274,372.947,-82.221,-176.182,9.313,148.785
C00708=1156.270,373.195,-82.257,-176.180,9.318,148.786
C00709=1156.266,373.442,-82.293,-176.178,9.321,148.786
C00710=1156.263,373.689,-82.329,-176.175,9.326,148.787
C00711=1156.258,373.936,-82.364,-176.174,9.330,148.787
C00712=1156.254,374.184,-82.400,-176.172,9.333,148.788
C00713=1156.250,374.431,-82.436,-176.169,9.338,148.788
C00714=1156.247,374.678,-82.472,-176.168,9.341,148.789
C00715=1156.243,374.926,-82.508,-176.166,9.345,148.789
C00716=1156.239,375.174,-82.544,-176.164,9.350,148.790
C00717=1156.235,375.421,-82.579,-176.163,9.354,148.791
C00718=1156.231,375.668,-82.616,-176.161,9.357,148.791
C00719=1156.228,375.916,-82.652,-176.159,9.361,148.792
C00720=1156.224,376.163,-82.687,-176.157,9.366,148.792
C00721=1156.219,376.410,-82.723,-176.155,9.369,148.793
C00722=1156.216,376.657,-82.759,-176.154,9.373,148.793
C00723=1156.211,376.905,-82.795,-176.152,9.377,148.794
C00724=1156.207,377.153,-82.831,-176.151,9.381,148.795
C00725=1156.204,377.400,-82.867,-176.149,9.385,148.795
C00726=1156.200,377.647,-82.903,-176.148,9.389,148.796
C00727=1156.196,377.894,-82.940,-176.146,9.393,148.796
C00728=1156.192,378.142,-82.976,-176.145,9.396,148.797
C00729=1156.188,378.390,-83.011,-176.143,9.400,148.798
C00730=1156.184,378.637,-83.048,-176.142,9.404,148.798
C00731=1156.181,378.884,-83.084,-176.141,9.408,148.799
C00732=1156.177,379.131,-83.120,-176.139,9.412,148.800
C00733=1156.173,379.379,-83.156,-176.138,9.416,148.800
C00734=1156.169,379.626,-83.192,-176.136,9.420,148.801
C00735=1156.165,379.874,-83.228,-176.135,9.424,148.801
C00736=1156.161,380.121,-83.264,-176.134,9.428,148.802
C00737=1156.157,380.368,-83.301,-176.133,9.431,148.803
C00738=1156.154,380.616,-83.336,-176.132,9.436,148.804
C00739=1156.150,380.863,-83.373,-176.130,9.439,148.804
C00740=1156.146,381.110,-83.409,-176.129,9.443,148.805
C00741=1156.142,381.358,-83.446,-176.129,9.447,148.806
C00742=1156.138,381.605,-83.482,-176.128,9.451,148.806
C00743=1156.134,381.852,-83.518,-176.127,9.454,148.807
C00744=1156.131,382.099,-83.554,-176.126,9.458,148.808
C00745=1156.126,382.347,-83.590,-176.125,9.462,148.809
C00746=1156.123,382.594,-83.627,-176.124,9.465,148.809
C00747=1156.119,382.842,-83.663,-176.123,9.469,148.810
C00748=1156.114,383.089,-83.700,-176.122,9.473,148.811
C00749=1156.111,383.336,-83.736,-176.122,9.476,148.812
C00750=1156.107,383.584,-83.772,-176.121,9.480,148.812
C00751=1156.103,383.830,-83.808,-176.120,9.484,148.813
C00752=1156.099,384.078,-83.845,-176.119,9.487,148.814
C00753=1156.096,384.325,-83.881,-176.119,9.490,148.815
C00754=1156.091,384.572,-83.918,-176.118,9.494,148.815
C00755=1156.088,384.819,-83.954,-176.118,9.498,148.816
C00756=1156.084,385.067,-83.990,-176.118,9.501,148.817
C00757=1156.080,385.314,-84.027,-176.118,9.504,148.818
C00758=1156.077,385.562,-84.064,-176.117,9.508,148.819
C00759=1156.072,385.810,-84.100,-176.117,9.511,148.819
C00760=1156.069,386.057,-84.136,-176.116,9.514,148.820
C00761=1156.065,386.304,-84.173,-176.116,9.518,148.821
C00762=1156.061,386.552,-84.209,-176.116,9.521,148.822
C00763=1156.057,386.798,-84.245,-176.116,9.524,148.822
C00764=1156.053,387.046,-84.282,-176.116,9.528,148.823
C00765=1156.049,387.293,-84.319,-176.116,9.530,148.824
C00766=1156.045,387.540,-84.354,-176.116,9.534,148.825
C00767=1156.041,387.787,-84.391,-176.116,9.537,148.826
C00768=1156.038,388.034,-84.428,-176.116,9.540,148.827
C00769=1156.034,388.282,-84.464,-176.116,9.543,148.827
C00770=1156.029,388.529,-84.501,-176.116,9.547,148.828
C00771=1156.027,388.777,-84.537,-176.116,9.549,148.829
C00772=1156.023,389.024,-84.574,-176.117,9.552,148.830
C00773=1156.018,389.271,-84.611,-176.117,9.555,148.831
C00774=1156.015,389.519,-84.646,-176.117,9.558,148.832
C00775=1156.011,389.766,-84.683,-176.117,9.561,148.832
C00776=1156.007,390.013,-84.720,-176.117,9.564,148.833
C00777=1156.003,390.260,-84.756,-176.118,9.567,148.834
C00778=1155.999,390.507,-84.793,-176.118,9.569,148.835
C00779=1155.995,390.755,-84.829,-176.119,9.572,148.836
C00780=1155.991,391.041,-84.872,-176.119,9.576,148.837
C00781=1155.986,391.327,-84.914,-176.119,9.579,148.838
C00782=1155.982,391.613,-84.957,-176.120,9.582,148.839
C00783=1155.977,391.899,-84.999,-176.121,9.585,148.840
C00784=1155.974,392.146,-85.035,-176.121,9.588,148.841
C00785=1155.970,392.393,-85.072,-176.121,9.590,148.841
C00786=1155.966,392.640,-85.109,-176.122,9.593,148.842
C00787=1155.963,392.889,-85.145,-176.122,9.596,148.843
C00788=1155.959,393.136,-85.182,-176.123,9.598,148.844
C00789=1155.955,393.383,-85.219,-176.124,9.600,148.845
C00790=1155.951,393.630,-85.255,-176.124,9.603,148.846
C00791=1155.947,393.877,-85.292,-176.125,9.605,148.846
C00792=1155.943,394.124,-85.329,-176.125,9.608,148.847
C00793=1155.939,394.372,-85.364,-176.126,9.611,148.848
C00794=1155.935,394.619,-85.401,-176.127,9.613,148.849
C00795=1155.932,394.867,-85.438,-176.127,9.615,148.850
C00796=1155.928,395.114,-85.474,-176.128,9.618,148.850
C00797=1155.924,395.361,-85.511,-176.129,9.620,148.851
C00798=1155.920,395.608,-85.548,-176.130,9.622,148.852
C00799=1155.916,395.855,-85.585,-176.130,9.625,148.853
C00800=1155.912,396.103,-85.621,-176.131,9.627,148.854
C00801=1155.908,396.350,-85.657,-176.131,9.630,148.854
C00802=1155.904,396.597,-85.694,-176.133,9.632,148.855
C00803=1155.901,396.844,-85.731,-176.134,9.634,148.856
C00804=1155.897,397.092,-85.768,-176.134,9.637,148.857
C00805=1155.893,397.339,-85.805,-176.135,9.638,148.858
C00806=1155.889,397.586,-85.842,-176.136,9.640,148.858
C00807=1155.886,397.834,-85.877,-176.136,9.643,148.859
C00808=1155.881,398.081,-85.914,-176.137,9.645,148.860
C00809=1155.877,398.328,-85.951,-176.138,9.647,148.861
C00810=1155.873,398.575,-85.988,-176.138,9.650,148.862
C00811=1155.870,398.822,-86.024,-176.140,9.652,148.862
C00812=1155.866,399.070,-86.061,-176.141,9.654,148.863
C00813=1155.862,399.317,-86.098,-176.141,9.656,148.864
C00814=1155.859,399.564,-86.134,-176.142,9.658,148.865
C00815=1155.855,399.811,-86.171,-176.143,9.660,148.865
C00816=1155.850,400.059,-86.207,-176.144,9.662,148.866
C00817=1155.846,400.306,-86.244,-176.144,9.664,148.867
C00818=1155.843,400.553,-86.280,-176.146,9.666,148.868
C00819=1155.840,400.801,-86.318,-176.147,9.668,148.869
C00820=1155.835,401.048,-86.354,-176.147,9.671,148.869
C00821=1155.831,401.296,-86.391,-176.148,9.673,148.870
C00822=1155.828,401.542,-86.428,-176.149,9.674,148.871
C00823=1155.824,401.790,-86.464,-176.150,9.677,148.872
C00824=1155.820,402.037,-86.501,-176.150,9.678,148.872
C00825=1155.816,402.284,-86.537,-176.151,9.680,148.873
C00826=1155.812,402.532,-86.574,-176.152,9.682,148.874
C00827=1155.809,402.779,-86.611,-176.153,9.684,148.874
C00828=1155.804,403.027,-86.648,-176.154,9.686,148.875
C00829=1155.801,403.274,-86.684,-176.154,9.688,148.876
C00830=1155.797,403.521,-86.721,-176.155,9.691,148.877
C00831=1155.793,403.768,-86.758,-176.156,9.692,148.877
C00832=1155.789,404.015,-86.795,-176.157,9.694,148.878
C00833=1155.785,404.262,-86.831,-176.158,9.696,148.879
C00834=1155.782,404.510,-86.868,-176.158,9.698,148.880
C00835=1155.778,404.758,-86.904,-176.159,9.700,148.880
C00836=1155.773,405.005,-86.941,-176.160,9.702,148.881
C00837=1155.770,405.252,-86.977,-176.161,9.703,148.882
C00838=1155.766,405.499,-87.014,-176.162,9.705,148.882
C00839=1155.762,405.746,-87.051,-176.163,9.707,148.883
C00840=1155.759,405.993,-87.087,-176.163,9.709,148.884
C00841=1155.755,406.241,-87.125,-176.164,9.711,148.884
C00842=1155.751,406.488,-87.161,-176.165,9.712,148.885
C00843=1155.747,406.735,-87.198,-176.166,9.715,148.886
C00844=1155.743,406.982,-87.235,-176.167,9.716,148.887
C00845=1155.739,407.229,-87.271,-176.167,9.718,148.887
C00846=1155.735,407.477,-87.308,-176.168,9.720,148.888
C00847=1155.731,407.724,-87.344,-176.169,9.722,148.889
C00848=1155.728,407.972,-87.381,-176.170,9.724,148.889
C00849=1155.724,408.219,-87.418,-176.171,9.725,148.890
C00850=1155.720,408.466,-87.455,-176.171,9.727,148.891
C00851=1155.716,408.713,-87.492,-176.172,9.729,148.891
C00852=1155.713,408.960,-87.528,-176.172,9.731,148.892
C00853=1155.708,409.208,-87.565,-176.173,9.733,148.893
C00854=1155.704,409.455,-87.602,-176.173,9.735,148.893
C00855=1155.701,409.703,-87.639,-176.174,9.737,148.894
C00856=1155.697,409.950,-87.675,-176.175,9.738,148.895
C00857=1155.693,410.197,-87.712,-176.176,9.740,148.895
C00858=1155.689,410.444,-87.749,-176.177,9.742,148.896
C00859=1155.685,410.691,-87.786,-176.177,9.744,148.897
C00860=1155.682,410.939,-87.821,-176.178,9.746,148.897
C00861=1155.677,411.186,-87.858,-176.179,9.747,148.898
C00862=1155.674,411.434,-87.895,-176.179,9.749,148.899
C00863=1155.670,411.681,-87.932,-176.180,9.751,148.899
C00864=1155.666,411.928,-87.968,-176.181,9.753,148.900
C00865=1155.662,412.175,-88.005,-176.181,9.754,148.901
C00866=1155.658,412.422,-88.042,-176.182,9.756,148.901
C00867=1155.654,412.669,-88.079,-176.183,9.758,148.902
C00868=1155.650,412.917,-88.116,-176.182,9.760,148.902
C00869=1155.647,413.164,-88.152,-176.183,9.762,148.903
C00870=1155.643,413.411,-88.189,-176.184,9.764,148.904
C00871=1155.639,413.658,-88.226,-176.184,9.765,148.904
C00872=1155.635,413.906,-88.263,-176.185,9.767,148.905
C00873=1155.632,414.153,-88.299,-176.186,9.769,148.906
C00874=1155.628,414.400,-88.336,-176.187,9.771,148.906
C00875=1155.624,414.648,-88.373,-176.187,9.772,148.907
C00876=1155.620,414.895,-88.410,-176.188,9.774,148.908
C00877=1155.617,415.142,-88.447,-176.188,9.777,148.908
C00878=1155.614,415.389,-88.483,-176.188,9.778,148.909
C00879=1155.612,415.637,-88.519,-176.189,9.780,148.909
C00880=1155.611,416.037,-88.578,-176.190,9.783,148.910
C00881=1155.612,416.435,-88.637,-176.191,9.785,148.911
C00882=1155.615,416.833,-88.695,-176.192,9.788,148.912
C00883=1155.621,417.231,-88.753,-176.192,9.791,148.913
C00884=1155.200,417.233,-88.801,-176.195,9.802,148.917
C00885=1155.195,416.832,-88.743,-176.195,9.799,148.916
C00886=1155.191,416.430,-88.683,-176.193,9.797,148.915
C00887=1155.190,416.028,-88.625,-176.193,9.794,148.914
C00888=1155.192,415.625,-88.565,-176.192,9.791,148.913
C00889=1155.194,415.378,-88.528,-176.191,9.789,148.912
C00890=1155.196,415.131,-88.492,-176.191,9.787,148.912
C00891=1155.199,414.883,-88.455,-176.190,9.786,148.911
C00892=1155.203,414.636,-88.418,-176.189,9.784,148.910
C00893=1155.207,414.389,-88.382,-176.189,9.781,148.910
C00894=1155.211,414.142,-88.345,-176.189,9.780,148.909
C00895=1155.215,413.895,-88.308,-176.188,9.778,148.908
C00896=1155.218,413.647,-88.271,-176.187,9.776,148.908
C00897=1155.222,413.400,-88.235,-176.186,9.774,148.907
C00898=1155.226,413.153,-88.198,-176.186,9.773,148.907
C00899=1155.230,412.905,-88.161,-176.186,9.771,148.906
C00900=1155.234,412.658,-88.124,-176.185,9.769,148.905
C00901=1155.237,412.411,-88.088,-176.184,9.768,148.905
C00902=1155.242,412.164,-88.052,-176.184,9.765,148.904
C00903=1155.245,411.916,-88.015,-176.183,9.763,148.903
C00904=1155.249,411.669,-87.978,-176.183,9.762,148.903
C00905=1155.253,411.421,-87.941,-176.182,9.760,148.902
C00906=1155.257,411.174,-87.905,-176.181,9.758,148.902
C00907=1155.261,410.927,-87.868,-176.181,9.756,148.901
C00908=1155.265,410.680,-87.831,-176.179,9.754,148.900
C00909=1155.269,410.432,-87.794,-176.179,9.753,148.899
C00910=1155.272,410.185,-87.757,-176.178,9.751,148.899
C00911=1155.276,409.938,-87.721,-176.177,9.749,148.898
C00912=1155.280,409.691,-87.684,-176.177,9.747,148.897
C00913=1155.284,409.444,-87.647,-176.176,9.746,148.897
C00914=1155.288,409.197,-87.611,-176.175,9.744,148.896
C00915=1155.292,408.950,-87.574,-176.175,9.742,148.896
C00916=1155.295,408.702,-87.536,-176.174,9.740,148.895
C00917=1155.299,408.455,-87.500,-176.173,9.739,148.894
C00918=1155.303,408.208,-87.463,-176.172,9.737,148.893
C00919=1155.307,407.960,-87.427,-176.172,9.735,148.893
C00920=1155.311,407.713,-87.390,-176.171,9.733,148.892
C00921=1155.315,407.465,-87.353,-176.170,9.731,148.891
C00922=1155.318,407.219,-87.317,-176.169,9.730,148.891
C00923=1155.322,406.971,-87.280,-176.168,9.727,148.890
C00924=1155.326,406.724,-87.243,-176.168,9.726,148.889
C00925=1155.330,406.476,-87.206,-176.168,9.723,148.889
C00926=1155.334,406.229,-87.170,-176.167,9.721,148.888
C00927=1155.338,405.982,-87.133,-176.166,9.719,148.887
C00928=1155.342,405.735,-87.096,-176.165,9.718,148.887
C00929=1155.345,405.487,-87.059,-176.164,9.716,148.886
C00930=1155.349,405.240,-87.023,-176.163,9.714,148.885
C00931=1155.353,404.993,-86.986,-176.163,9.712,148.884
C00932=1155.357,404.746,-86.949,-176.162,9.710,148.884
C00933=1155.361,404.498,-86.913,-176.161,9.708,148.883
C00934=1155.365,404.251,-86.877,-176.160,9.706,148.882
C00935=1155.369,404.004,-86.840,-176.159,9.705,148.882
C00936=1155.372,403.756,-86.803,-176.158,9.703,148.881
C00937=1155.376,403.509,-86.766,-176.158,9.701,148.880
C00938=1155.380,403.262,-86.729,-176.156,9.699,148.879
C00939=1155.384,403.015,-86.693,-176.156,9.697,148.879
C00940=1155.388,402.768,-86.656,-176.155,9.695,148.878
C00941=1155.392,402.521,-86.619,-176.154,9.693,148.877
C00942=1155.395,402.274,-86.583,-176.153,9.692,148.877
C00943=1155.399,402.026,-86.545,-176.152,9.689,148.876
C00944=1155.403,401.779,-86.509,-176.151,9.688,148.875
C00945=1155.407,401.531,-86.472,-176.151,9.685,148.874
C00946=1155.411,401.284,-86.436,-176.150,9.683,148.873
C00947=1155.415,401.037,-86.399,-176.149,9.681,148.873
C00948=1155.419,400.789,-86.362,-176.148,9.679,148.872
C00949=1155.422,400.543,-86.326,-176.147,9.677,148.871
C00950=1155.426,400.295,-86.289,-176.147,9.675,148.871
C00951=1155.430,400.048,-86.252,-176.145,9.673,148.870
C00952=1155.434,399.800,-86.215,-176.145,9.671,148.869
C00953=1155.437,399.553,-86.179,-176.144,9.669,148.868
C00954=1155.441,399.306,-86.142,-176.143,9.667,148.867
C00955=1155.446,399.058,-86.106,-176.142,9.665,148.867
C00956=1155.450,398.811,-86.069,-176.141,9.663,148.866
C00957=1155.453,398.564,-86.033,-176.141,9.660,148.865
C00958=1155.457,398.316,-85.996,-176.140,9.658,148.864
C00959=1155.461,398.069,-85.959,-176.139,9.656,148.863
C00960=1155.465,397.822,-85.922,-176.138,9.654,148.863
C00961=1155.468,397.575,-85.886,-176.138,9.652,148.862
C00962=1155.472,397.328,-85.849,-176.137,9.650,148.861
C00963=1155.476,397.081,-85.812,-176.135,9.648,148.860
C00964=1155.480,396.833,-85.776,-176.135,9.645,148.859
C00965=1155.484,396.586,-85.740,-176.134,9.643,148.859
C00966=1155.488,396.338,-85.702,-176.134,9.640,148.858
C00967=1155.492,396.091,-85.665,-176.133,9.638,148.857
C00968=1155.495,395.844,-85.629,-176.132,9.636,148.856
C00969=1155.499,395.597,-85.592,-176.131,9.633,148.855
C00970=1155.503,395.350,-85.555,-176.130,9.631,148.854
C00971=1155.507,395.103,-85.519,-176.130,9.629,148.854
C00972=1155.511,394.855,-85.483,-176.129,9.627,148.853
C00973=1155.515,394.608,-85.446,-176.128,9.624,148.852
C00974=1155.519,394.360,-85.409,-176.128,9.622,148.851
C00975=1155.522,394.113,-85.373,-176.127,9.619,148.850
C00976=1155.526,393.866,-85.336,-176.127,9.616,148.850
C00977=1155.530,393.619,-85.299,-176.126,9.614,148.849
C00978=1155.533,393.372,-85.263,-176.125,9.612,148.848
C00979=1155.538,393.124,-85.227,-176.125,9.609,148.847
C00980=1155.542,392.877,-85.190,-176.124,9.607,148.846
C00981=1155.546,392.630,-85.153,-176.123,9.604,148.845
C00982=1155.549,392.382,-85.116,-176.123,9.601,148.845
C00983=1155.553,392.135,-85.079,-176.123,9.598,148.844
C00984=1155.557,391.888,-85.043,-176.122,9.596,148.843
C00985=1155.561,391.602,-85.001,-176.121,9.593,148.842
C00986=1155.565,391.316,-84.958,-176.121,9.590,148.841
C00987=1155.570,391.030,-84.916,-176.120,9.587,148.840
C00988=1155.575,390.743,-84.874,-176.120,9.583,148.839
C00989=1155.578,390.496,-84.837,-176.120,9.580,148.838
C00990=1155.582,390.249,-84.801,-176.119,9.577,148.837
C00991=1155.586,390.002,-84.764,-176.119,9.575,148.837
C00992=1155.590,389.755,-84.727,-176.119,9.572,148.836
C00993=1155.594,389.507,-84.691,-176.118,9.569,148.835
C00994=1155.598,389.260,-84.654,-176.118,9.567,148.834
C00995=1155.602,389.013,-84.618,-176.118,9.563,148.833
C00996=1155.605,388.765,-84.581,-176.117,9.560,148.832
C00997=1155.609,388.518,-84.544,-176.117,9.557,148.832
C00998=1155.613,388.270,-84.509,-176.117,9.554,148.831
C00999=1155.617,388.023,-84.472,-176.117,9.551,148.830
C01000=1155.621,387.776,-84.435,-176.117,9.548,148.829
C01001=1155.624,387.529,-84.399,-176.117,9.545,148.828
C01002=1155.629,387.281,-84.362,-176.117,9.542,148.827
C01003=1155.632,387.034,-84.326,-176.117,9.539,148.827
C01004=1155.636,386.787,-84.289,-176.118,9.535,148.826
C01005=1155.640,386.540,-84.252,-176.117,9.532,148.825
C01006=1155.644,386.293,-84.217,-176.117,9.529,148.824
C01007=1155.647,386.045,-84.180,-176.118,9.526,148.823
C01008=1155.652,385.798,-84.143,-176.118,9.522,148.823
C01009=1155.655,385.551,-84.107,-176.118,9.519,148.822
C01010=1155.659,385.303,-84.070,-176.118,9.516,148.821
C01011=1155.663,385.056,-84.034,-176.119,9.513,148.820
C01012=1155.667,384.809,-83.997,-176.119,9.509,148.820
C01013=1155.671,384.561,-83.961,-176.120,9.505,148.819
C01014=1155.674,384.314,-83.925,-176.121,9.502,148.818
C01015=1155.679,384.067,-83.888,-176.121,9.498,148.817
C01016=1155.682,383.819,-83.853,-176.122,9.495,148.816
C01017=1155.686,383.572,-83.816,-176.122,9.492,148.816
C01018=1155.690,383.325,-83.779,-176.123,9.487,148.815
C01019=1155.694,383.077,-83.743,-176.124,9.484,148.814
C01020=1155.698,382.830,-83.706,-176.124,9.481,148.813
C01021=1155.702,382.583,-83.671,-176.125,9.476,148.812
C01022=1155.706,382.336,-83.634,-176.126,9.473,148.812
C01023=1155.709,382.089,-83.598,-176.127,9.469,148.811
C01024=1155.714,381.841,-83.562,-176.127,9.466,148.810
C01025=1155.717,381.594,-83.525,-176.129,9.462,148.810
C01026=1155.721,381.346,-83.489,-176.130,9.458,148.809
C01027=1155.725,381.099,-83.453,-176.131,9.454,148.808
C01028=1155.729,380.851,-83.416,-176.132,9.450,148.808
C01029=1155.732,380.604,-83.380,-176.133,9.446,148.807
C01030=1155.736,380.356,-83.344,-176.134,9.443,148.806
C01031=1155.740,380.109,-83.308,-176.135,9.439,148.806
C01032=1155.744,379.862,-83.271,-176.137,9.435,148.805
C01033=1155.748,379.615,-83.236,-176.138,9.431,148.804
C01034=1155.752,379.367,-83.200,-176.139,9.427,148.803
C01035=1155.756,379.121,-83.163,-176.141,9.423,148.803
C01036=1155.760,378.873,-83.127,-176.142,9.419,148.802
C01037=1155.764,378.626,-83.091,-176.144,9.415,148.802
C01038=1155.768,378.378,-83.055,-176.145,9.412,148.801
C01039=1155.771,378.131,-83.018,-176.146,9.408,148.800
C01040=1155.775,377.884,-82.983,-176.148,9.404,148.800
C01041=1155.779,377.636,-82.947,-176.149,9.400,148.799
C01042=1155.783,377.389,-82.911,-176.151,9.396,148.798
C01043=1155.787,377.141,-82.874,-176.152,9.392,148.798
C01044=1155.791,376.894,-82.838,-176.154,9.388,148.797
C01045=1155.795,376.647,-82.802,-176.155,9.384,148.797
C01046=1155.799,376.399,-82.766,-176.157,9.381,148.796
C01047=1155.802,376.152,-82.730,-176.159,9.376,148.796
C01048=1155.806,375.904,-82.694,-176.161,9.372,148.795
C01049=1155.810,375.657,-82.658,-176.163,9.368,148.794
C01050=1155.813,375.410,-82.622,-176.164,9.365,148.794
C01051=1155.818,375.162,-82.586,-176.166,9.360,148.793
C01052=1155.822,374.915,-82.551,-176.168,9.356,148.793
C01053=1155.826,374.668,-82.515,-176.169,9.352,148.792
C01054=1155.830,374.421,-82.478,-176.172,9.348,148.792
C01055=1155.833,374.173,-82.443,-176.174,9.344,148.791
C01056=1155.837,373.926,-82.407,-176.175,9.341,148.791
C01057=1155.842,373.678,-82.371,-176.178,9.336,148.790
C01058=1155.845,373.430,-82.336,-176.180,9.333,148.790
C01059=1155.849,373.183,-82.299,-176.181,9.329,148.789
C01060=1155.852,372.936,-82.264,-176.183,9.324,148.789
C01061=1155.857,372.689,-82.228,-176.185,9.321,148.788
C01062=1155.861,372.441,-82.193,-176.188,9.316,148.788
C01063=1155.865,372.194,-82.157,-176.189,9.312,148.787
C01064=1155.868,371.946,-82.121,-176.192,9.308,148.787
C01065=1155.873,371.699,-82.085,-176.194,9.304,148.786
C01066=1155.876,371.451,-82.050,-176.196,9.300,148.786
C01067=1155.880,371.204,-82.014,-176.198,9.296,148.785
C01068=1155.884,370.957,-81.979,-176.200,9.292,148.785
C01069=1155.889,370.709,-81.943,-176.202,9.288,148.784
C01070=1155.892,370.461,-81.907,-176.205,9.284,148.784
C01071=1155.896,370.214,-81.872,-176.207,9.280,148.784
C01072=1155.900,369.966,-81.836,-176.209,9.276,148.783
C01073=1155.904,369.720,-81.801,-176.211,9.272,148.783
C01074=1155.907,369.472,-81.766,-176.214,9.268,148.782
C01075=1155.912,369.224,-81.729,-176.216,9.265,148.782
C01076=1155.916,368.977,-81.694,-176.218,9.260,148.781
C01077=1155.919,368.729,-81.658,-176.221,9.256,148.781
C01078=1155.923,368.483,-81.623,-176.223,9.252,148.781
C01079=1155.927,368.235,-81.588,-176.226,9.248,148.780
C01080=1155.931,367.988,-81.552,-176.227,9.245,148.780
C01081=1155.934,367.740,-81.516,-176.230,9.240,148.779
C01082=1155.939,367.493,-81.482,-176.233,9.236,148.779
C01083=1155.943,367.245,-81.446,-176.235,9.232,148.779
C01084=1155.947,366.997,-81.410,-176.237,9.228,148.778
C01085=1155.951,366.750,-81.375,-176.239,9.225,148.778
C01086=1155.955,366.503,-81.340,-176.242,9.220,148.778
C01087=1155.959,366.255,-81.305,-176.244,9.216,148.777
C01088=1155.963,366.007,-81.269,-176.247,9.213,148.777
C01089=1155.967,365.725,-81.229,-176.250,9.207,148.776
C01090=1155.971,365.442,-81.189,-176.253,9.203,148.776
C01091=1155.976,365.159,-81.149,-176.255,9.199,148.776
C01092=1155.980,364.876,-81.108,-176.258,9.195,148.775
C01093=1155.984,364.629,-81.073,-176.260,9.190,148.775
C01094=1155.988,364.381,-81.038,-176.263,9.186,148.774
C01095=1155.992,364.133,-81.002,-176.265,9.183,148.774
C01096=1155.996,363.887,-80.967,-176.268,9.179,148.774
C01097=1156.000,363.639,-80.932,-176.271,9.174,148.773
C01098=1156.004,363.391,-80.897,-176.273,9.171,148.773
C01099=1156.008,363.144,-80.862,-176.275,9.167,148.773
C01100=1156.012,362.896,-80.827,-176.278,9.163,148.773
C01101=1156.015,362.648,-80.793,-176.280,9.159,148.772
C01102=1156.020,362.402,-80.757,-176.283,9.155,148.772
C01103=1156.023,362.154,-80.722,-176.285,9.151,148.772
C01104=1156.027,361.906,-80.687,-176.288,9.147,148.771
C01105=1156.031,361.659,-80.652,-176.290,9.144,148.771
C01106=1156.035,361.411,-80.617,-176.293,9.140,148.771
C01107=1156.040,361.164,-80.582,-176.295,9.135,148.770
C01108=1156.043,360.916,-80.548,-176.298,9.132,148.770
C01109=1156.047,360.668,-80.513,-176.300,9.128,148.769
C01110=1156.051,360.421,-80.478,-176.303,9.124,148.769
C01111=1156.055,360.173,-80.443,-176.305,9.120,148.769
C01112=1156.059,359.926,-80.407,-176.308,9.116,148.768
C01113=1156.063,359.679,-80.373,-176.310,9.113,148.768
C01114=1156.067,359.431,-80.339,-176.313,9.108,148.768
C01115=1156.071,359.184,-80.303,-176.315,9.105,148.768
C01116=1156.075,358.936,-80.268,-176.318,9.101,148.767
C01117=1156.079,358.688,-80.234,-176.321,9.097,148.767
C01118=1156.082,358.441,-80.199,-176.323,9.093,148.767
C01119=1156.086,358.193,-80.164,-176.326,9.089,148.766
C01120=1156.091,357.946,-80.130,-176.328,9.086,148.766
C01121=1156.095,357.697,-80.095,-176.330,9.081,148.766
C01122=1156.098,357.451,-80.060,-176.333,9.078,148.765
C01123=1156.102,357.203,-80.026,-176.336,9.074,148.765
C01124=1156.107,356.955,-79.991,-176.338,9.071,148.765
C01125=1156.110,356.708,-79.957,-176.340,9.066,148.765
C01126=1156.114,356.461,-79.922,-176.343,9.063,148.764
C01127=1156.118,356.213,-79.887,-176.345,9.059,148.764
C01128=1156.122,355.966,-79.853,-176.347,9.055,148.764
C01129=1156.126,355.717,-79.818,-176.350,9.051,148.763
C01130=1156.131,355.470,-79.784,-176.353,9.048,148.763
C01131=1156.134,355.222,-79.749,-176.355,9.043,148.763
C01132=1156.139,354.975,-79.715,-176.357,9.040,148.762
C01133=1156.142,354.727,-79.680,-176.360,9.036,148.762
C01134=1156.146,354.480,-79.646,-176.363,9.033,148.762
C01135=1156.150,354.232,-79.611,-176.365,9.028,148.762
C01136=1156.154,353.985,-79.577,-176.367,9.025,148.761
C01137=1156.158,353.738,-79.542,-176.370,9.021,148.761
C01138=1156.162,353.490,-79.508,-176.372,9.017,148.761
C01139=1156.166,353.242,-79.474,-176.375,9.013,148.760
C01140=1156.170,352.994,-79.439,-176.377,9.010,148.760
C01141=1156.174,352.747,-79.405,-176.380,9.006,148.760
C01142=1156.178,352.498,-79.371,-176.382,9.002,148.760
C01143=1156.182,352.251,-79.337,-176.385,8.998,148.759
C01144=1156.187,352.004,-79.302,-176.387,8.995,148.759
C01145=1156.190,351.756,-79.268,-176.390,8.991,148.759
C01146=1156.194,351.509,-79.234,-176.392,8.988,148.759
C01147=1156.198,351.261,-79.200,-176.395,8.983,148.758
C01148=1156.202,351.013,-79.165,-176.397,8.980,148.758
C01149=1156.206,350.766,-79.131,-176.400,8.976,148.758
C01150=1156.210,350.518,-79.096,-176.402,8.973,148.757
C01151=1156.214,350.270,-79.063,-176.405,8.968,148.757
C01152=1156.218,350.022,-79.028,-176.407,8.965,148.757
C01153=1156.222,349.775,-78.995,-176.410,8.962,148.757
C01154=1156.227,349.528,-78.960,-176.412,8.957,148.756
C01155=1156.230,349.280,-78.926,-176.415,8.954,148.756
C01156=1156.234,349.032,-78.893,-176.417,8.950,148.756
C01157=1156.239,348.785,-78.858,-176.420,8.946,148.755
C01158=1156.242,348.537,-78.824,-176.422,8.942,148.755
C01159=1156.247,348.289,-78.790,-176.425,8.939,148.755
C01160=1156.250,348.042,-78.756,-176.428,8.935,148.755
C01161=1156.254,347.794,-78.722,-176.430,8.932,148.754
C01162=1156.259,347.546,-78.688,-176.432,8.928,148.754
C01163=1156.262,347.299,-78.654,-176.435,8.924,148.754
C01164=1156.266,347.051,-78.620,-176.437,8.921,148.754
C01165=1156.270,346.803,-78.586,-176.440,8.917,148.753
C01166=1156.274,346.556,-78.553,-176.442,8.913,148.753
C01167=1156.278,346.309,-78.519,-176.445,8.909,148.753
C01168=1156.282,346.060,-78.485,-176.447,8.906,148.752
C01169=1156.286,345.813,-78.451,-176.450,8.902,148.752
C01170=1156.290,345.565,-78.418,-176.452,8.898,148.752
C01171=1156.295,345.318,-78.383,-176.454,8.895,148.752
C01172=1156.299,345.069,-78.350,-176.457,8.891,148.752
C01173=1156.302,344.822,-78.316,-176.460,8.888,148.751
C01174=1156.307,344.574,-78.282,-176.463,8.884,148.751
C01175=1156.311,344.327,-78.248,-176.465,8.880,148.751
C01176=1156.315,344.079,-78.215,-176.467,8.876,148.750
C01177=1156.318,343.832,-78.181,-176.470,8.873,148.750
C01178=1156.323,343.584,-78.147,-176.472,8.869,148.750
C01179=1156.327,343.336,-78.114,-176.475,8.865,148.750
C01180=1156.331,343.088,-78.080,-176.477,8.862,148.750
C01181=1156.335,342.840,-78.046,-176.480,8.858,148.749
C01182=1156.339,342.593,-78.013,-176.482,8.855,148.749
C01183=1156.344,342.345,-77.979,-176.485,8.851,148.749
C01184=1156.348,342.097,-77.946,-176.488,8.847,148.749
C01185=1156.351,341.850,-77.912,-176.490,8.844,148.748
C01186=1156.355,341.602,-77.878,-176.492,8.839,148.748
C01187=1156.359,341.354,-77.845,-176.495,8.836,148.748
C01188=1156.363,341.106,-77.812,-176.497,8.833,148.748
C01189=1156.368,340.859,-77.777,-176.500,8.829,148.747
C01190=1156.372,340.611,-77.744,-176.502,8.825,148.747
C01191=1156.376,340.363,-77.711,-176.505,8.821,148.747
C01192=1156.380,340.115,-77.678,-176.507,8.818,148.747
C01193=1156.384,339.835,-77.640,-176.510,8.814,148.746
C01194=1156.389,339.556,-77.603,-176.513,8.810,148.746
C01195=1156.394,339.276,-77.564,-176.516,8.806,148.746
C01196=1156.398,338.996,-77.527,-176.519,8.802,148.746
C01197=1156.402,338.748,-77.493,-176.521,8.798,148.745
C01198=1156.406,338.500,-77.460,-176.524,8.795,148.745
C01199=1156.410,338.253,-77.426,-176.526,8.791,148.745
C01200=1156.414,338.005,-77.393,-176.529,8.788,148.745
C01201=1156.419,337.758,-77.360,-176.532,8.784,148.745
C01202=1156.423,337.510,-77.327,-176.534,8.780,148.744
C01203=1156.426,337.262,-77.293,-176.536,8.777,148.744
C01204=1156.430,337.014,-77.260,-176.539,8.773,148.744
C01205=1156.435,336.766,-77.227,-176.541,8.770,148.744
C01206=1156.439,336.518,-77.194,-176.544,8.766,148.743
C01207=1156.443,336.271,-77.161,-176.547,8.762,148.743
C01208=1156.447,336.023,-77.128,-176.549,8.759,148.743
C01209=1156.451,335.775,-77.094,-176.552,8.755,148.743
C01210=1156.455,335.527,-77.061,-176.554,8.752,148.743
C01211=1156.459,335.280,-77.028,-176.556,8.748,148.742
C01212=1156.463,335.032,-76.996,-176.559,8.744,148.742
C01213=1156.467,334.785,-76.962,-176.562,8.741,148.742
C01214=1156.471,334.537,-76.929,-176.564,8.738,148.742
C01215=1156.475,334.289,-76.896,-176.567,8.734,148.741
C01216=1156.479,334.041,-76.863,-176.569,8.730,148.741
C01217=1156.484,333.793,-76.831,-176.572,8.727,148.741
C01218=1156.488,333.545,-76.797,-176.574,8.723,148.741
C01219=1156.492,333.298,-76.764,-176.577,8.720,148.741
C01220=1156.495,333.050,-76.732,-176.579,8.716,148.740
C01221=1156.500,332.802,-76.698,-176.582,8.712,148.740
C01222=1156.504,332.555,-76.665,-176.584,8.709,148.740
C01223=1156.508,332.306,-76.633,-176.587,8.706,148.740
C01224=1156.512,332.059,-76.600,-176.589,8.702,148.740
C01225=1156.516,331.811,-76.567,-176.592,8.698,148.739
C01226=1156.520,331.563,-76.534,-176.594,8.695,148.739
C01227=1156.524,331.315,-76.502,-176.597,8.691,148.739
C01228=1156.528,331.067,-76.468,-176.600,8.688,148.739
C01229=1156.533,330.820,-76.435,-176.602,8.685,148.739
C01230=1156.536,330.572,-76.403,-176.605,8.681,148.738
C01231=1156.540,330.324,-76.370,-176.607,8.677,148.738
C01232=1156.545,330.076,-76.337,-176.609,8.674,148.738
C01233=1156.549,329.828,-76.305,-176.612,8.670,148.738
C01234=1156.552,329.580,-76.272,-176.615,8.667,148.738
C01235=1156.557,329.333,-76.239,-176.617,8.663,148.737
C01236=1156.561,329.084,-76.207,-176.620,8.659,148.737
C01237=1156.566,328.837,-76.174,-176.622,8.656,148.737
C01238=1156.569,328.589,-76.142,-176.625,8.653,148.737
C01239=1156.574,328.341,-76.109,-176.627,8.650,148.737
C01240=1156.578,328.093,-76.076,-176.630,8.646,148.737
C01241=1156.581,327.846,-76.044,-176.632,8.642,148.736
C01242=1156.586,327.597,-76.011,-176.635,8.639,148.736
C01243=1156.589,327.350,-75.979,-176.638,8.635,148.736
C01244=1156.594,327.102,-75.946,-176.640,8.632,148.736
C01245=1156.598,326.854,-75.913,-176.642,8.628,148.736
C01246=1156.602,326.607,-75.882,-176.646,8.625,148.736
C01247=1156.606,326.359,-75.848,-176.648,8.621,148.735
C01248=1156.611,326.110,-75.816,-176.650,8.618,148.735
C01249=1156.614,325.863,-75.783,-176.653,8.615,148.735
C01250=1156.619,325.615,-75.751,-176.655,8.611,148.735
C01251=1156.622,325.367,-75.719,-176.658,8.607,148.734
C01252=1156.627,325.120,-75.686,-176.660,8.605,148.735
C01253=1156.631,324.872,-75.655,-176.663,8.600,148.734
C01254=1156.635,324.624,-75.621,-176.666,8.597,148.734
C01255=1156.639,324.376,-75.590,-176.668,8.594,148.734
C01256=1156.643,324.127,-75.557,-176.670,8.591,148.734
C01257=1156.647,323.879,-75.525,-176.673,8.586,148.733
C01258=1156.651,323.632,-75.492,-176.676,8.584,148.733
C01259=1156.655,323.384,-75.461,-176.678,8.580,148.733
C01260=1156.660,323.136,-75.428,-176.681,8.576,148.733
C01261=1156.663,322.889,-75.396,-176.683,8.573,148.733
C01262=1156.667,322.640,-75.363,-176.686,8.570,148.733
C01263=1156.672,322.393,-75.332,-176.689,8.567,148.733
C01264=1156.676,322.145,-75.299,-176.691,8.563,148.732
C01265=1156.680,321.897,-75.267,-176.694,8.559,148.732
C01266=1156.684,321.649,-75.234,-176.696,8.556,148.732
C01267=1156.688,321.401,-75.203,-176.698,8.553,148.732
C01268=1156.692,321.153,-75.171,-176.702,8.549,148.732
C01269=1156.696,320.905,-75.139,-176.704,8.546,148.732
C01270=1156.700,320.657,-75.107,-176.706,8.542,148.731
C01271=1156.705,320.409,-75.075,-176.709,8.538,148.731
C01272=1156.709,320.161,-75.043,-176.711,8.535,148.731
C01273=1156.713,319.913,-75.011,-176.714,8.532,148.731
C01274=1156.718,319.666,-74.979,-176.717,8.529,148.731
C01275=1156.721,319.418,-74.946,-176.719,8.525,148.731
C01276=1156.725,319.170,-74.914,-176.722,8.521,148.730
C01277=1156.729,318.922,-74.882,-176.725,8.518,148.730
C01278=1156.734,318.675,-74.850,-176.727,8.515,148.730
C01279=1156.737,318.426,-74.819,-176.730,8.511,148.730
C01280=1156.742,318.178,-74.786,-176.732,8.508,148.730
C01281=1156.746,317.931,-74.755,-176.735,8.505,148.730
C01282=1156.750,317.683,-74.723,-176.737,8.501,148.730
C01283=1156.754,317.434,-74.691,-176.739,8.498,148.729
C01284=1156.759,317.186,-74.660,-176.743,8.494,148.729
C01285=1156.762,316.938,-74.628,-176.745,8.491,148.729
C01286=1156.766,316.690,-74.596,-176.747,8.488,148.729
C01287=1156.771,316.443,-74.564,-176.750,8.485,148.729
C01288=1156.775,316.195,-74.532,-176.753,8.481,148.729
C01289=1156.779,315.947,-74.500,-176.755,8.478,148.729
C01290=1156.783,315.699,-74.469,-176.758,8.474,148.728
C01291=1156.788,315.450,-74.437,-176.760,8.471,148.728
C01292=1156.792,315.203,-74.406,-176.763,8.467,148.728
C01293=1156.796,314.955,-74.374,-176.766,8.464,148.728
C01294=1156.799,314.707,-74.342,-176.768,8.461,148.728
C01295=1156.804,314.460,-74.310,-176.771,8.458,148.728
C01296=1156.808,314.211,-74.279,-176.773,8.454,148.728
C01297=1156.813,313.934,-74.243,-176.776,8.450,148.727
C01298=1156.818,313.656,-74.208,-176.779,8.446,148.727
C01299=1156.822,313.379,-74.172,-176.782,8.442,148.727
C01300=1156.827,313.102,-74.137,-176.784,8.439,148.727
C01301=1156.831,312.853,-74.106,-176.788,8.435,148.727
C01302=1156.835,312.606,-74.074,-176.790,8.432,148.727
C01303=1156.839,312.358,-74.042,-176.792,8.429,148.727
C01304=1156.844,312.110,-74.012,-176.795,8.426,148.727
C01305=1156.847,311.862,-73.980,-176.797,8.423,148.726
C01306=1156.852,311.614,-73.949,-176.800,8.418,148.726
C01307=1156.856,311.366,-73.917,-176.803,8.415,148.726
C01308=1156.860,311.119,-73.886,-176.805,8.412,148.726
C01309=1156.864,310.870,-73.855,-176.808,8.409,148.726
C01310=1156.868,310.623,-73.823,-176.810,8.406,148.726
C01311=1156.872,310.374,-73.792,-176.813,8.402,148.726
C01312=1156.877,310.126,-73.760,-176.816,8.399,148.726
C01313=1156.881,309.878,-73.729,-176.818,8.396,148.725
C01314=1156.886,309.630,-73.697,-176.821,8.392,148.725
C01315=1156.890,309.382,-73.666,-176.823,8.389,148.725
C01316=1156.894,309.134,-73.635,-176.826,8.385,148.725
C01317=1156.898,308.886,-73.604,-176.829,8.382,148.725
C01318=1156.902,308.638,-73.572,-176.831,8.379,148.725
C01319=1156.906,308.390,-73.541,-176.834,8.376,148.725
C01320=1156.910,308.143,-73.510,-176.836,8.373,148.725
C01321=1156.914,307.894,-73.479,-176.839,8.370,148.725
C01322=1156.918,307.646,-73.448,-176.842,8.365,148.724
C01323=1156.922,307.398,-73.416,-176.844,8.362,148.724
C01324=1156.927,307.150,-73.386,-176.847,8.359,148.724
C01325=1156.931,306.902,-73.355,-176.849,8.356,148.724
C01326=1156.935,306.654,-73.323,-176.852,8.353,148.724
C01327=1156.940,306.406,-73.292,-176.854,8.350,148.724
C01328=1156.944,306.157,-73.261,-176.857,8.346,148.724
C01329=1156.948,305.910,-73.230,-176.860,8.343,148.724
C01330=1156.952,305.661,-73.199,-176.862,8.340,148.724
C01331=1156.957,305.413,-73.168,-176.865,8.336,148.723
C01332=1156.961,305.166,-73.138,-176.868,8.333,148.724
C01333=1156.964,304.918,-73.106,-176.870,8.330,148.723
C01334=1156.969,304.670,-73.075,-176.873,8.326,148.723
C01335=1156.973,304.422,-73.044,-176.875,8.323,148.723
C01336=1156.977,304.173,-73.013,-176.878,8.320,148.723
C01337=1156.982,303.925,-72.982,-176.881,8.317,148.723
C01338=1156.985,303.677,-72.951,-176.883,8.314,148.723
C01339=1156.990,303.429,-72.920,-176.886,8.311,148.723
C01340=1156.994,303.182,-72.890,-176.888,8.306,148.723
C01341=1156.998,302.933,-72.858,-176.891,8.304,148.723
C01342=1157.003,302.685,-72.828,-176.894,8.300,148.722
C01343=1157.007,302.437,-72.797,-176.896,8.297,148.722
C01344=1157.011,302.189,-72.766,-176.899,8.294,148.722
C01345=1157.015,301.941,-72.736,-176.901,8.291,148.722
C01346=1157.020,301.693,-72.705,-176.904,8.288,148.722
C01347=1157.023,301.444,-72.674,-176.907,8.284,148.722
C01348=1157.028,301.196,-72.644,-176.909,8.281,148.722
C01349=1157.033,300.948,-72.613,-176.912,8.277,148.722
C01350=1157.036,300.701,-72.583,-176.914,8.274,148.722
C01351=1157.040,300.452,-72.551,-176.917,8.271,148.722
C01352=1157.045,300.204,-72.521,-176.919,8.268,148.722
C01353=1157.049,299.956,-72.491,-176.922,8.265,148.721
C01354=1157.053,299.708,-72.459,-176.925,8.261,148.721
C01355=1157.058,299.460,-72.429,-176.927,8.258,148.721
C01356=1157.061,299.212,-72.398,-176.930,8.255,148.721
C01357=1157.066,298.964,-72.368,-176.932,8.252,148.721
C01358=1157.070,298.716,-72.337,-176.935,8.249,148.721
C01359=1157.074,298.468,-72.306,-176.938,8.245,148.721
C01360=1157.079,298.220,-72.276,-176.940,8.242,148.721
C01361=1157.083,297.972,-72.245,-176.943,8.238,148.721
C01362=1157.087,297.723,-72.215,-176.946,8.235,148.721
C01363=1157.091,297.475,-72.184,-176.948,8.232,148.721
C01364=1157.095,297.227,-72.154,-176.951,8.229,148.721
C01365=1157.100,296.980,-72.123,-176.954,8.226,148.721
C01366=1157.103,296.731,-72.093,-176.956,8.223,148.721
C01367=1157.108,296.483,-72.063,-176.959,8.220,148.721
C01368=1157.112,296.235,-72.033,-176.961,8.217,148.720
C01369=1157.117,295.987,-72.002,-176.964,8.214,148.720
C01370=1157.121,295.739,-71.971,-176.967,8.210,148.720
C01371=1157.125,295.490,-71.941,-176.970,8.207,148.720
C01372=1157.129,295.242,-71.911,-176.972,8.203,148.720
C01373=1157.133,294.994,-71.880,-176.975,8.200,148.720
C01374=1157.137,294.746,-71.851,-176.977,8.197,148.720
C01375=1157.142,294.498,-71.820,-176.980,8.194,148.720
C01376=1157.146,294.251,-71.790,-176.982,8.191,148.720
C01377=1157.150,294.001,-71.760,-176.985,8.188,148.720
C01378=1157.154,293.754,-71.729,-176.988,8.185,148.720
C01379=1157.159,293.505,-71.699,-176.990,8.182,148.720
C01380=1157.163,293.257,-71.669,-176.993,8.178,148.720
C01381=1157.167,293.009,-71.638,-176.996,8.175,148.720
C01382=1157.172,292.761,-71.609,-176.998,8.172,148.720
C01383=1157.176,292.514,-71.579,-177.001,8.169,148.720
C01384=1157.180,292.264,-71.548,-177.003,8.166,148.719
C01385=1157.184,292.017,-71.518,-177.006,8.163,148.719
C01386=1157.189,291.768,-71.488,-177.008,8.159,148.719
C01387=1157.193,291.520,-71.458,-177.011,8.156,148.719
C01388=1157.197,291.272,-71.429,-177.014,8.153,148.719
C01389=1157.201,291.024,-71.398,-177.016,8.150,148.719
C01390=1157.205,290.776,-71.368,-177.019,8.147,148.719
C01391=1157.209,290.528,-71.338,-177.022,8.143,148.719
C01392=1157.214,290.280,-71.308,-177.025,8.140,148.719
C01393=1157.218,290.031,-71.279,-177.027,8.137,148.719
C01394=1157.222,289.783,-71.248,-177.030,8.134,148.719
C01395=1157.227,289.534,-71.218,-177.032,8.131,148.719
C01396=1157.231,289.287,-71.188,-177.035,8.128,148.719
C01397=1157.235,289.039,-71.158,-177.037,8.125,148.719
C01398=1157.239,288.790,-71.129,-177.040,8.122,148.719
C01399=1157.244,288.542,-71.098,-177.043,8.119,148.719
C01400=1157.248,288.294,-71.069,-177.045,8.115,148.719
C01401=1157.252,288.019,-71.035,-177.049,8.112,148.719
C01402=1157.257,287.744,-71.003,-177.051,8.109,148.719
C01403=1157.262,287.469,-70.970,-177.054,8.105,148.719
C01404=1157.267,287.194,-70.937,-177.057,8.102,148.719
C01405=1157.271,286.946,-70.907,-177.060,8.099,148.719
C01406=1157.275,286.698,-70.877,-177.062,8.095,148.718
C01407=1157.280,286.449,-70.847,-177.065,8.093,148.718
C01408=1157.284,286.201,-70.818,-177.068,8.090,148.719
C01409=1157.288,285.953,-70.788,-177.071,8.085,148.718
C01410=1157.292,285.704,-70.759,-177.073,8.082,148.718
C01411=1157.297,285.456,-70.729,-177.076,8.080,148.718
C01412=1157.300,285.209,-70.699,-177.078,8.076,148.718
C01413=1157.305,284.960,-70.669,-177.081,8.073,148.718
C01414=1157.310,284.712,-70.640,-177.084,8.070,148.718
C01415=1157.314,284.463,-70.610,-177.086,8.067,148.718
C01416=1157.318,284.215,-70.581,-177.089,8.064,148.718
C01417=1157.322,283.967,-70.551,-177.092,8.061,148.718
C01418=1157.326,283.719,-70.522,-177.094,8.058,148.718
C01419=1157.330,283.470,-70.492,-177.097,8.055,148.718
C01420=1157.335,283.222,-70.463,-177.100,8.052,148.718
C01421=1157.339,282.974,-70.434,-177.102,8.049,148.718
C01422=1157.343,282.726,-70.404,-177.105,8.046,148.718
C01423=1157.349,282.478,-70.374,-177.107,8.043,148.718
C01424=1157.353,282.229,-70.345,-177.110,8.040,148.718
C01425=1157.357,281.981,-70.316,-177.113,8.037,148.718
C01426=1157.361,281.733,-70.286,-177.115,8.034,148.718
C01427=1157.365,281.485,-70.257,-177.118,8.031,148.718
C01428=1157.369,281.236,-70.227,-177.121,8.028,148.718
C01429=1157.374,280.988,-70.198,-177.123,8.024,148.718
C01430=1157.378,280.740,-70.168,-177.126,8.021,148.718
C01431=1157.383,280.492,-70.139,-177.129,8.019,148.718
C01432=1157.387,280.244,-70.110,-177.131,8.016,148.718
C01433=1157.391,279.995,-70.081,-177.134,8.012,148.718
C01434=1157.395,279.747,-70.052,-177.136,8.009,148.718
C01435=1157.400,279.499,-70.022,-177.139,8.006,148.718
C01436=1157.403,279.251,-69.993,-177.142,8.003,148.718
C01437=1157.407,279.002,-69.964,-177.144,8.000,148.718
C01438=1157.412,278.755,-69.935,-177.147,7.997,148.718
C01439=1157.416,278.506,-69.906,-177.150,7.994,148.718
C01440=1157.421,278.258,-69.876,-177.153,7.991,148.718
C01441=1157.425,278.009,-69.847,-177.155,7.988,148.718
C01442=1157.429,277.761,-69.818,-177.158,7.985,148.718
C01443=1157.434,277.512,-69.789,-177.160,7.982,148.718
C01444=1157.438,277.265,-69.760,-177.163,7.979,148.718
C01445=1157.442,277.017,-69.731,-177.165,7.976,148.718
C01446=1157.446,276.768,-69.702,-177.168,7.973,148.718
C01447=1157.450,276.520,-69.673,-177.171,7.970,148.718
C01448=1157.455,276.271,-69.643,-177.174,7.967,148.718
C01449=1157.460,276.023,-69.615,-177.177,7.964,148.718
C01450=1157.464,275.775,-69.585,-177.179,7.961,148.718
C01451=1157.467,275.527,-69.557,-177.182,7.958,148.718
C01452=1157.472,275.278,-69.528,-177.184,7.955,148.718
C01453=1157.477,275.030,-69.499,-177.187,7.952,148.718
C01454=1157.481,274.782,-69.470,-177.190,7.949,148.718
C01455=1157.485,274.533,-69.441,-177.192,7.946,148.718
C01456=1157.489,274.285,-69.412,-177.195,7.943,148.718
C01457=1157.494,274.037,-69.383,-177.198,7.940,148.718
C01458=1157.498,273.789,-69.354,-177.200,7.937,148.718
C01459=1157.502,273.540,-69.325,-177.203,7.934,148.718
C01460=1157.506,273.293,-69.297,-177.206,7.931,148.718
C01461=1157.511,273.044,-69.268,-177.208,7.928,148.718
C01462=1157.515,272.796,-69.238,-177.211,7.925,148.718
C01463=1157.519,272.547,-69.210,-177.214,7.922,148.718
C01464=1157.524,272.299,-69.182,-177.217,7.919,148.718
C01465=1157.528,272.051,-69.152,-177.219,7.916,148.718
C01466=1157.533,271.802,-69.124,-177.222,7.913,148.718
C01467=1157.537,271.554,-69.095,-177.224,7.910,148.718
C01468=1157.541,271.305,-69.067,-177.227,7.907,148.718
C01469=1157.545,271.058,-69.038,-177.230,7.904,148.718
C01470=1157.550,270.809,-69.009,-177.233,7.901,148.718
C01471=1157.554,270.560,-68.981,-177.236,7.898,148.718
C01472=1157.558,270.312,-68.952,-177.238,7.895,148.718
C01473=1157.563,270.064,-68.923,-177.241,7.892,148.718
C01474=1157.567,269.815,-68.895,-177.243,7.889,148.718
C01475=1157.571,269.567,-68.866,-177.246,7.886,148.718
C01476=1157.576,269.319,-68.837,-177.249,7.883,148.718
C01477=1157.580,269.071,-68.809,-177.252,7.880,148.718
C01478=1157.585,268.823,-68.781,-177.254,7.877,148.718
C01479=1157.589,268.574,-68.752,-177.257,7.874,148.718
C01480=1157.593,268.326,-68.723,-177.260,7.871,148.718
C01481=1157.598,268.077,-68.695,-177.262,7.868,148.718
C01482=1157.601,267.829,-68.667,-177.265,7.865,148.718
C01483=1157.606,267.581,-68.638,-177.267,7.863,148.718
C01484=1157.610,267.332,-68.610,-177.270,7.860,148.718
C01485=1157.614,267.084,-68.581,-177.273,7.857,148.719
C01486=1157.619,266.836,-68.553,-177.276,7.854,148.719
C01487=1157.623,266.587,-68.524,-177.278,7.851,148.719
C01488=1157.628,266.339,-68.496,-177.281,7.848,148.719
C01489=1157.632,266.090,-68.468,-177.284,7.845,148.719
C01490=1157.636,265.842,-68.440,-177.286,7.842,148.719
C01491=1157.641,265.594,-68.411,-177.289,7.839,148.719
C01492=1157.645,265.346,-68.383,-177.292,7.836,148.719
C01493=1157.650,265.097,-68.355,-177.294,7.833,148.719
C01494=1157.654,264.848,-68.327,-177.297,7.830,148.719
C01495=1157.659,264.600,-68.298,-177.300,7.827,148.719
C01496=1157.662,264.351,-68.270,-177.303,7.824,148.719
C01497=1157.667,264.104,-68.242,-177.305,7.821,148.719
C01498=1157.671,263.855,-68.214,-177.308,7.819,148.719
C01499=1157.676,263.607,-68.186,-177.310,7.816,148.719
C01500=1157.680,263.358,-68.157,-177.313,7.813,148.719
C01501=1157.684,263.110,-68.129,-177.316,7.810,148.719
C01502=1157.688,262.861,-68.101,-177.319,7.807,148.719
C01503=1157.693,262.613,-68.073,-177.322,7.804,148.719
C01504=1157.697,262.365,-68.045,-177.324,7.801,148.719
C01505=1157.702,262.092,-68.014,-177.327,7.798,148.720
C01506=1157.707,261.819,-67.984,-177.330,7.795,148.720
C01507=1157.712,261.546,-67.952,-177.333,7.792,148.720
C01508=1157.717,261.272,-67.921,-177.336,7.789,148.720
C01509=1157.721,261.023,-67.893,-177.339,7.786,148.720
C01510=1157.725,260.775,-67.866,-177.341,7.783,148.720
C01511=1157.730,260.526,-67.837,-177.344,7.780,148.720
C01512=1157.734,260.279,-67.809,-177.347,7.777,148.720
C01513=1157.738,260.030,-67.781,-177.350,7.774,148.720
C01514=1157.742,259.782,-67.754,-177.353,7.771,148.720
C01515=1157.747,259.533,-67.726,-177.354,7.769,148.720
C01516=1157.751,259.285,-67.697,-177.357,7.766,148.720
C01517=1157.755,259.037,-67.670,-177.360,7.763,148.720
C01518=1157.760,258.788,-67.642,-177.363,7.760,148.720
C01519=1157.765,258.539,-67.614,-177.365,7.757,148.720
C01520=1157.769,258.292,-67.586,-177.368,7.754,148.720
C01521=1157.773,258.042,-67.559,-177.371,7.751,148.720
C01522=1157.777,257.795,-67.531,-177.374,7.748,148.720
C01523=1157.781,257.546,-67.503,-177.376,7.745,148.720
C01524=1157.787,257.297,-67.475,-177.379,7.743,148.720
C01525=1157.791,257.049,-67.447,-177.381,7.740,148.721
C01526=1157.795,256.801,-67.419,-177.384,7.737,148.721
C01527=1157.799,256.552,-67.392,-177.387,7.734,148.721
C01528=1157.804,256.304,-67.364,-177.390,7.731,148.721
C01529=1157.808,256.055,-67.337,-177.392,7.728,148.721
C01530=1157.812,255.807,-67.309,-177.396,7.725,148.721
C01531=1157.817,255.558,-67.282,-177.398,7.723,148.721
C01532=1157.821,255.310,-67.253,-177.401,7.720,148.721
C01533=1157.826,255.062,-67.226,-177.403,7.717,148.721
C01534=1157.830,254.814,-67.199,-177.406,7.715,148.721
C01535=1157.834,254.564,-67.171,-177.409,7.712,148.721
C01536=1157.839,254.316,-67.143,-177.412,7.709,148.721
C01537=1157.843,254.068,-67.116,-177.414,7.706,148.722
C01538=1157.847,253.819,-67.088,-177.417,7.703,148.722
C01539=1157.852,253.571,-67.061,-177.420,7.700,148.722
C01540=1157.856,253.323,-67.033,-177.422,7.698,148.722
C01541=1157.861,253.075,-67.006,-177.425,7.695,148.722
C01542=1157.864,252.826,-66.978,-177.428,7.692,148.722
C01543=1157.869,252.577,-66.951,-177.431,7.689,148.722
C01544=1157.874,252.329,-66.924,-177.433,7.686,148.722
C01545=1157.877,252.080,-66.896,-177.436,7.683,148.722
C01546=1157.882,251.832,-66.869,-177.438,7.681,148.722
C01547=1157.887,251.583,-66.842,-177.441,7.678,148.722
C01548=1157.891,251.335,-66.814,-177.444,7.675,148.722
C01549=1157.895,251.086,-66.786,-177.447,7.672,148.722
C01550=1157.900,250.838,-66.759,-177.449,7.669,148.722
C01551=1157.904,250.590,-66.732,-177.453,7.666,148.723
C01552=1157.909,250.341,-66.705,-177.455,7.664,148.723
C01553=1157.914,250.093,-66.678,-177.458,7.661,148.723
C01554=1157.918,249.844,-66.650,-177.460,7.658,148.723
C01555=1157.922,249.596,-66.622,-177.463,7.656,148.723
C01556=1157.927,249.347,-66.595,-177.466,7.653,148.723
C01557=1157.931,249.099,-66.568,-177.469,7.650,148.723
C01558=1157.935,248.851,-66.542,-177.471,7.647,148.723
C01559=1157.939,248.601,-66.514,-177.474,7.645,148.723
C01560=1157.944,248.353,-66.487,-177.476,7.642,148.723
C01561=1157.948,248.105,-66.459,-177.479,7.639,148.723
C01562=1157.953,247.857,-66.432,-177.482,7.636,148.724
C01563=1157.958,247.608,-66.405,-177.485,7.633,148.724
C01564=1157.962,247.360,-66.378,-177.487,7.631,148.724
C01565=1157.966,247.111,-66.351,-177.490,7.628,148.724
C01566=1157.970,246.862,-66.324,-177.493,7.625,148.724
C01567=1157.975,246.614,-66.297,-177.496,7.622,148.724
C01568=1157.979,246.365,-66.270,-177.498,7.619,148.724
C01569=1157.984,246.117,-66.243,-177.501,7.617,148.724
C01570=1157.988,245.869,-66.217,-177.504,7.614,148.725
C01571=1157.993,245.620,-66.190,-177.507,7.612,148.725
C01572=1157.997,245.371,-66.162,-177.509,7.609,148.725
C01573=1158.001,245.122,-66.135,-177.512,7.606,148.725
C01574=1158.005,244.874,-66.109,-177.515,7.603,148.725
C01575=1158.010,244.626,-66.082,-177.517,7.601,148.725
C01576=1158.015,244.377,-66.055,-177.520,7.598,148.725
C01577=1158.019,244.129,-66.028,-177.523,7.595,148.725
C01578=1158.023,243.881,-66.001,-177.526,7.592,148.725
C01579=1158.028,243.632,-65.974,-177.528,7.590,148.726
C01580=1158.033,243.384,-65.947,-177.531,7.587,148.726
C01581=1158.036,243.135,-65.920,-177.534,7.584,148.726
C01582=1158.041,242.887,-65.893,-177.536,7.581,148.726
C01583=1158.045,242.637,-65.867,-177.539,7.578,148.726
C01584=1158.049,242.389,-65.840,-177.542,7.576,148.726
C01585=1158.054,242.140,-65.813,-177.545,7.574,148.726
C01586=1158.059,241.892,-65.786,-177.547,7.571,148.726
C01587=1158.063,241.644,-65.760,-177.550,7.568,148.726
C01588=1158.067,241.395,-65.733,-177.553,7.565,148.726
C01589=1158.072,241.146,-65.706,-177.555,7.563,148.727
C01590=1158.076,240.898,-65.680,-177.558,7.560,148.727
C01591=1158.081,240.649,-65.653,-177.561,7.557,148.727
C01592=1158.085,240.401,-65.626,-177.564,7.554,148.727
C01593=1158.090,240.152,-65.600,-177.566,7.552,148.727
C01594=1158.094,239.904,-65.573,-177.569,7.549,148.727
C01595=1158.098,239.655,-65.546,-177.572,7.546,148.727
C01596=1158.103,239.406,-65.520,-177.575,7.543,148.728
C01597=1158.107,239.158,-65.494,-177.577,7.541,148.728
C01598=1158.112,238.910,-65.466,-177.580,7.538,148.728
C01599=1158.116,238.661,-65.441,-177.583,7.535,148.728
C01600=1158.121,238.412,-65.414,-177.586,7.533,148.728
C01601=1158.125,238.164,-65.387,-177.588,7.531,148.728
C01602=1158.130,237.915,-65.361,-177.591,7.528,148.728
C01603=1158.134,237.667,-65.334,-177.594,7.525,148.728
C01604=1158.138,237.418,-65.307,-177.596,7.522,148.728
C01605=1158.142,237.170,-65.282,-177.599,7.520,148.729
C01606=1158.148,236.922,-65.255,-177.602,7.517,148.729
C01607=1158.152,236.673,-65.229,-177.605,7.514,148.729
C01608=1158.157,236.424,-65.202,-177.607,7.511,148.729
C01609=1158.161,236.153,-65.174,-177.611,7.509,148.729
C01610=1158.166,235.881,-65.145,-177.613,7.506,148.729
C01611=1158.170,235.609,-65.116,-177.616,7.503,148.729
C01612=1158.176,235.337,-65.087,-177.619,7.500,148.730
C01613=1158.180,235.089,-65.061,-177.622,7.497,148.730
C01614=1158.185,234.840,-65.034,-177.624,7.495,148.730
C01615=1158.189,234.591,-65.009,-177.627,7.492,148.730
C01616=1158.193,234.343,-64.982,-177.630,7.490,148.730
C01617=1158.198,234.094,-64.956,-177.633,7.487,148.730
C01618=1158.202,233.846,-64.929,-177.635,7.485,148.730
C01619=1158.206,233.597,-64.904,-177.638,7.482,148.731
C01620=1158.211,233.348,-64.877,-177.641,7.479,148.731
C01621=1158.216,233.100,-64.851,-177.644,7.477,148.731
C01622=1158.220,232.852,-64.826,-177.646,7.474,148.731
C01623=1158.225,232.603,-64.798,-177.650,7.471,148.731
C01624=1158.229,232.354,-64.773,-177.652,7.468,148.731
C01625=1158.233,232.106,-64.747,-177.655,7.466,148.732
C01626=1158.238,231.856,-64.721,-177.657,7.463,148.732
C01627=1158.242,231.608,-64.694,-177.661,7.461,148.732
C01628=1158.247,231.360,-64.669,-177.663,7.459,148.732
C01629=1158.252,231.111,-64.642,-177.666,7.456,148.732
C01630=1158.256,230.863,-64.616,-177.668,7.453,148.732
C01631=1158.260,230.614,-64.590,-177.672,7.450,148.732
C01632=1158.264,230.365,-64.564,-177.674,7.448,148.733
C01633=1158.270,230.117,-64.538,-177.677,7.445,148.733
C01634=1158.274,229.868,-64.513,-177.680,7.443,148.733
C01635=1158.278,229.620,-64.486,-177.682,7.440,148.733
C01636=1158.282,229.371,-64.460,-177.685,7.438,148.733
C01637=1158.286,229.122,-64.435,-177.688,7.435,148.733
C01638=1158.292,228.874,-64.409,-177.690,7.433,148.734
C01639=1158.296,228.625,-64.383,-177.693,7.430,148.734
C01640=1158.300,228.376,-64.357,-177.696,7.427,148.734
C01641=1158.305,228.127,-64.332,-177.698,7.425,148.734
C01642=1158.309,227.879,-64.306,-177.701,7.422,148.734
C01643=1158.314,227.631,-64.279,-177.704,7.419,148.734
C01644=1158.318,227.382,-64.253,-177.707,7.418,148.735
C01645=1158.322,227.133,-64.228,-177.709,7.415,148.735
C01646=1158.327,226.885,-64.202,-177.712,7.412,148.735
C01647=1158.332,226.636,-64.176,-177.715,7.410,148.735
C01648=1158.336,226.387,-64.151,-177.718,7.407,148.735
C01649=1158.341,226.139,-64.125,-177.720,7.404,148.735
C01650=1158.345,225.891,-64.100,-177.723,7.402,148.736
C01651=1158.350,225.641,-64.073,-177.726,7.399,148.736
C01652=1158.354,225.393,-64.047,-177.729,7.396,148.736
C01653=1158.359,225.145,-64.022,-177.731,7.395,148.736
C01654=1158.363,224.896,-63.996,-177.734,7.392,148.736
C01655=1158.367,224.647,-63.971,-177.737,7.389,148.736
C01656=1158.372,224.398,-63.946,-177.740,7.387,148.737
C01657=1158.377,224.149,-63.920,-177.742,7.384,148.737
C01658=1158.381,223.901,-63.894,-177.745,7.381,148.737
C01659=1158.386,223.652,-63.869,-177.748,7.379,148.737
C01660=1158.390,223.404,-63.843,-177.751,7.376,148.737
C01661=1158.394,223.155,-63.817,-177.753,7.373,148.737
C01662=1158.399,222.907,-63.792,-177.756,7.372,148.738
C01663=1158.403,222.657,-63.767,-177.759,7.369,148.738
C01664=1158.408,222.409,-63.742,-177.761,7.367,148.738
C01665=1158.413,222.160,-63.716,-177.764,7.364,148.738
C01666=1158.417,221.912,-63.690,-177.767,7.361,148.738
C01667=1158.422,221.664,-63.665,-177.769,7.359,148.738
C01668=1158.426,221.414,-63.640,-177.773,7.356,148.739
C01669=1158.430,221.165,-63.614,-177.775,7.353,148.739
C01670=1158.435,220.917,-63.589,-177.778,7.352,148.739
C01671=1158.439,220.668,-63.563,-177.781,7.349,148.739
C01672=1158.445,220.420,-63.538,-177.783,7.347,148.739
C01673=1158.448,220.171,-63.513,-177.786,7.344,148.740
C01674=1158.452,219.922,-63.487,-177.789,7.341,148.740
C01675=1158.457,219.674,-63.463,-177.792,7.339,148.740
C01676=1158.462,219.425,-63.437,-177.794,7.336,148.740
C01677=1158.466,219.177,-63.412,-177.797,7.333,148.740
C01678=1158.471,218.927,-63.386,-177.800,7.332,148.740
C01679=1158.476,218.679,-63.361,-177.803,7.329,148.741
C01680=1158.479,218.431,-63.336,-177.805,7.327,148.741
C01681=1158.484,218.181,-63.311,-177.808,7.324,148.741
C01682=1158.489,217.933,-63.286,-177.811,7.321,148.741
C01683=1158.493,217.684,-63.260,-177.814,7.319,148.741
C01684=1158.498,217.436,-63.235,-177.816,7.316,148.742
C01685=1158.503,217.186,-63.210,-177.819,7.315,148.742
C01686=1158.507,216.938,-63.185,-177.822,7.312,148.742
C01687=1158.511,216.690,-63.160,-177.824,7.310,148.742
C01688=1158.516,216.441,-63.135,-177.827,7.307,148.742
C01689=1158.520,216.192,-63.109,-177.830,7.304,148.742
C01690=1158.525,215.944,-63.085,-177.833,7.302,148.743
C01691=1158.529,215.694,-63.060,-177.835,7.299,148.743
C01692=1158.534,215.446,-63.035,-177.838,7.297,148.743
C01693=1158.538,215.197,-63.010,-177.841,7.295,148.743
C01694=1158.543,214.949,-62.985,-177.843,7.293,148.743
C01695=1158.547,214.700,-62.960,-177.846,7.290,148.744
C01696=1158.552,214.451,-62.934,-177.849,7.287,148.744
C01697=1158.556,214.202,-62.909,-177.852,7.285,148.744
C01698=1158.561,213.954,-62.885,-177.855,7.282,148.744
C01699=1158.565,213.705,-62.859,-177.857,7.280,148.744
C01700=1158.570,213.456,-62.835,-177.860,7.278,148.745
C01701=1158.574,213.208,-62.810,-177.862,7.275,148.745
C01702=1158.579,212.959,-62.785,-177.866,7.273,148.745
C01703=1158.584,212.710,-62.760,-177.868,7.270,148.745
C01704=1158.588,212.461,-62.736,-177.871,7.268,148.746
C01705=1158.593,212.213,-62.710,-177.874,7.265,148.746
C01706=1158.597,211.963,-62.685,-177.876,7.263,148.746
C01707=1158.601,211.715,-62.661,-177.879,7.261,148.746
C01708=1158.606,211.467,-62.636,-177.882,7.259,148.746
C01709=1158.610,211.218,-62.612,-177.885,7.256,148.747
C01710=1158.615,210.969,-62.587,-177.887,7.254,148.747
C01711=1158.620,210.720,-62.562,-177.890,7.251,148.747
C01712=1158.624,210.472,-62.537,-177.892,7.249,148.747
C01713=1158.629,210.201,-62.511,-177.896,7.246,148.747
C01714=1158.634,209.930,-62.484,-177.899,7.244,148.748
C01715=1158.639,209.660,-62.457,-177.902,7.241,148.748
C01716=1158.644,209.389,-62.430,-177.905,7.238,148.748
C01717=1158.649,209.140,-62.406,-177.907,7.236,148.748
C01718=1158.653,208.893,-62.381,-177.910,7.234,148.749
C01719=1158.657,208.643,-62.356,-177.913,7.232,148.749
C01720=1158.662,208.395,-62.332,-177.916,7.229,148.749
C01721=1158.667,208.146,-62.307,-177.918,7.227,148.749
C01722=1158.671,207.897,-62.283,-177.921,7.224,148.750
C01723=1158.676,207.648,-62.258,-177.923,7.222,148.750
C01724=1158.680,207.400,-62.234,-177.927,7.220,148.750
C01725=1158.685,207.150,-62.209,-177.929,7.217,148.750
C01726=1158.689,206.902,-62.185,-177.932,7.215,148.750
C01727=1158.694,206.653,-62.160,-177.935,7.212,148.750
C01728=1158.698,206.404,-62.136,-177.938,7.210,148.751
C01729=1158.703,206.155,-62.111,-177.940,7.207,148.751
C01730=1158.708,205.907,-62.087,-177.943,7.206,148.751
C01731=1158.713,205.658,-62.062,-177.946,7.203,148.751
C01732=1158.716,205.409,-62.038,-177.949,7.201,148.752
C01733=1158.722,205.160,-62.013,-177.951,7.198,148.752
C01734=1158.726,204.912,-61.989,-177.954,7.196,148.752
C01735=1158.730,204.663,-61.965,-177.957,7.193,148.752
C01736=1158.735,204.414,-61.940,-177.959,7.191,148.753
C01737=1158.739,204.166,-61.916,-177.962,7.188,148.753
C01738=1158.744,203.917,-61.892,-177.965,7.187,148.753
C01739=1158.749,203.667,-61.867,-177.967,7.185,148.753
C01740=1158.753,203.419,-61.843,-177.970,7.182,148.754
C01741=1158.757,203.171,-61.819,-177.973,7.180,148.754
C01742=1158.762,202.922,-61.795,-177.976,7.177,148.754
C01743=1158.766,202.673,-61.770,-177.979,7.176,148.754
C01744=1158.771,202.424,-61.746,-177.981,7.173,148.754
C01745=1158.776,202.175,-61.722,-177.984,7.171,148.755
C01746=1158.780,201.927,-61.698,-177.987,7.168,148.755
C01747=1158.785,201.678,-61.674,-177.989,7.166,148.755
C01748=1158.789,201.429,-61.649,-177.992,7.163,148.755
C01749=1158.794,201.180,-61.626,-177.995,7.162,148.756
C01750=1158.798,200.931,-61.601,-177.998,7.159,148.756
C01751=1158.803,200.683,-61.577,-178.000,7.157,148.756
C01752=1158.808,200.434,-61.553,-178.004,7.154,148.756
C01753=1158.812,200.184,-61.529,-178.006,7.152,148.757
C01754=1158.817,199.936,-61.505,-178.009,7.150,148.757
C01755=1158.821,199.688,-61.481,-178.011,7.147,148.757
C01756=1158.826,199.438,-61.457,-178.014,7.146,148.757
C01757=1158.831,199.190,-61.433,-178.017,7.143,148.757
C01758=1158.835,198.941,-61.409,-178.019,7.141,148.758
C01759=1158.839,198.692,-61.385,-178.023,7.138,148.758
C01760=1158.844,198.443,-61.361,-178.025,7.136,148.758
C01761=1158.849,198.195,-61.336,-178.028,7.134,148.759
C01762=1158.853,197.945,-61.313,-178.030,7.132,148.759
C01763=1158.858,197.697,-61.289,-178.034,7.129,148.759
C01764=1158.863,197.448,-61.266,-178.036,7.127,148.759
C01765=1158.867,197.200,-61.241,-178.039,7.125,148.760
C01766=1158.872,196.951,-61.218,-178.042,7.123,148.760
C01767=1158.876,196.702,-61.194,-178.044,7.120,148.760
C01768=1158.881,196.452,-61.170,-178.047,7.118,148.760
C01769=1158.885,196.204,-61.146,-178.049,7.116,148.760
C01770=1158.890,195.955,-61.122,-178.053,7.113,148.761
C01771=1158.894,195.706,-61.098,-178.055,7.111,148.761
C01772=1158.899,195.457,-61.075,-178.058,7.109,148.761
C01773=1158.903,195.209,-61.051,-178.061,7.107,148.762
C01774=1158.908,194.960,-61.027,-178.063,7.105,148.762
C01775=1158.913,194.711,-61.003,-178.066,7.102,148.762
C01776=1158.917,194.462,-60.980,-178.069,7.100,148.762
C01777=1158.922,194.213,-60.957,-178.072,7.097,148.763
C01778=1158.926,193.965,-60.933,-178.075,7.096,148.763
C01779=1158.931,193.716,-60.909,-178.077,7.094,148.763
C01780=1158.935,193.467,-60.885,-178.080,7.091,148.763
C01781=1158.940,193.218,-60.862,-178.083,7.089,148.764
C01782=1158.946,192.969,-60.838,-178.085,7.086,148.764
C01783=1158.950,192.721,-60.814,-178.088,7.085,148.764
C01784=1158.955,192.472,-60.790,-178.091,7.083,148.765
C01785=1158.959,192.223,-60.767,-178.094,7.080,148.765
C01786=1158.963,191.975,-60.743,-178.096,7.078,148.765
C01787=1158.968,191.726,-60.720,-178.100,7.076,148.765
C01788=1158.972,191.476,-60.697,-178.102,7.073,148.765
C01789=1158.977,191.227,-60.673,-178.104,7.072,148.766
C01790=1158.982,190.979,-60.649,-178.107,7.069,148.766
C01791=1158.986,190.730,-60.626,-178.110,7.067,148.766
C01792=1158.991,190.481,-60.603,-178.113,7.064,148.767
C01793=1158.996,190.232,-60.579,-178.115,7.062,148.767
C01794=1159.000,189.984,-60.555,-178.118,7.061,148.767
C01795=1159.005,189.734,-60.532,-178.121,7.058,148.767
C01796=1159.009,189.485,-60.508,-178.124,7.056,148.768
C01797=1159.014,189.236,-60.485,-178.127,7.053,148.768
C01798=1159.019,188.987,-60.462,-178.129,7.052,148.768
C01799=1159.024,188.738,-60.438,-178.132,7.049,148.768
C01800=1159.027,188.490,-60.415,-178.135,7.047,148.769
C01801=1159.032,188.241,-60.392,-178.138,7.045,148.769
C01802=1159.037,187.992,-60.368,-178.140,7.043,148.769
C01803=1159.041,187.743,-60.345,-178.143,7.040,148.770
C01804=1159.046,187.494,-60.321,-178.146,7.039,148.770
C01805=1159.051,187.245,-60.298,-178.149,7.036,148.770
C01806=1159.056,186.997,-60.275,-178.151,7.034,148.770
C01807=1159.060,186.748,-60.252,-178.154,7.032,148.771
C01808=1159.065,186.499,-60.229,-178.157,7.029,148.771
C01809=1159.069,186.250,-60.206,-178.159,7.028,148.771
